// oaksLibrary/fbPumpMotion
// Block för global pumpmotion. V i blocket sätter internt i blocket den globala variabeln oaksGVL.bPumpMotion. 
// oaksGVL.bPumpMotion finns knuten i fbMotor och aktiverar pumpmotion om bPumpmotionConfig i respektive fbMotor-instans är till.
FUNCTION_BLOCK fbPumpMotion
VAR_INPUT
END_VAR
VAR_OUTPUT
	{attribute 'OPC.UA.DA' := '1'}
	V AT %M*  : BOOL; //Pumpmotion aktiv~wp:[trendoptions]i:14400, t:1
	{attribute 'OPC.UA.DA' := '1'}
	PV AT %M*  : STRING; //Dag för motionering~wp:
	{attribute 'OPC.UA.DA' := '1'}
	PV1 AT %M* : INT; //Tid för motionering~wp:[format]00:00
END_VAR
VAR
	stTime		: tc2_ba.TIMESTRUCT;
	nActualDayCase	: INT;
	nActualHour 	: INT;
	nActualMinute 	: INT;
	
	FB_BA_GetTime01 : tc2_ba.FB_BA_GetTime; 
	FB_BA_ExtTiSt01 : tc2_ba.FB_BA_ExtTiSt;	
	
	itemp : INT;
	nTime : INT; // Internvariabel aktuell tid (nActualHour+nActualMinute)
	
	bDay : BOOL; // Internvariabel blir TRUE om inställd dag är lika med aktuell dag
	bTime : BOOL; // Internvariabel blir TRUE om inställd tid är lika med aktuell tid
END_VAR
VAR_INPUT PERSISTENT
	{attribute 'OPC.UA.DA' := '1'}
	SP1 AT %M*  : INT:=1; //Dag för pumpmotion (0 = Söndag 1 = Måndag 2 = Tisdag..6 = Lördag~wp:
	{attribute 'OPC.UA.DA' := '1'}
	SP2 AT %M*  : INT:=1000; //Tid för pumpmotion~wp:[format]00:00[engmin]0[engmax]2400
END_VAR

	IF SP1 < 0 OR  SP1>6 THEN
		SP1 := 1;
	END_IF
	
	IF SP2 < 0 OR  SP2>2359 THEN
		SP2 := 1200;
	END_IF
	
	

	FB_BA_GetTime01(bEn :=TRUE);	
	stTime := FB_BA_GetTime01.stSysTi;

	nActualDayCase :=WORD_TO_INT (stTime.wDayOfWeek);
	nActualHour :=WORD_TO_INT (stTime.wHour)*100;
	nActualMinute :=WORD_TO_INT (stTime.wMinute);
	
	// nActualHour+nActualMinute
	
	nTime := nActualHour+nActualMinute;
	
	bDay := nActualDayCase = SP1;
	bTime := nTime = SP2;
	
	
	V := bDay AND bTime;
	
	oaksGVL.bPumpMotion := V;
	
	//För visning i Webport	
	PV1:= SP2;

	CASE SP1 OF
		0: PV:= 'Söndag';
		1: PV:= 'Måndag';
		2: PV:= 'Tisdag';
		3: PV:= 'Onsdag';
		4: PV:= 'Torsdag';
		5: PV:= 'Fredag';
		6: PV:= 'Lördag';
	END_CASE

END_FUNCTION_BLOCK

// oaksLibrary/Brand/fbFireDamperOneInput
//Funktionsblock för styrning av brandspjäll med stängt indikering (stänger på fjäder). 
FUNCTION_BLOCK fbFireDamperOneInput EXTENDS fbDigitalSignalLogic
VAR_INPUT
bMotion : BOOL; //Motionskörning
{attribute 'OPC.UA.DA' := '1'}
V2 AT %I* : BOOL; //Stängindikering~wp:[trendoptions]i:14400, t:1
END_VAR
VAR_OUTPUT
	{attribute 'OPC.UA.DA' := '1'}
	AL AT %M* : BOOL; //Spjällfel~wp:
	{attribute 'OPC.UA.DA' := '1'}
	PV4 AT %M* : BOOL; //Motionskörning aktiv~wp:[trendoptions]i:14400, t:1
END_VAR
VAR
	SR_1: SR;
	fbStartPulse: TP; // Startpuls	
	fbMotionTime: TP; // Håller en puls under motionskörning
	fbStopMotion: F_TRIG;
	TON_1: TON;
	bAlarm: BOOL;
END_VAR

SUPER^();
//Aktivera motionering på positiv flank (SET)
fbStartPulse(IN:= bMotion, PT:= T#1S, Q=> , ET=> ); //Startar en puls

//Hållkrets
SR_1(
SET1:= fbStartPulse.Q, 
RESET:= fbStopMotion.Q OR V2, 
Q1=> PV4
);

//Avaktivera motionering (RESET)
fbMotionTime(IN:= fbStartPulse.Q, PT:= T#180S, Q=> , ET=> ); //Startar en puls
fbStopMotion(CLK:= fbMotionTime.Q OR V2, Q=> ); // Reset då pulstid gått ut eller stängtindikering gått till

//Utgång
CMD := bSafe AND bStart AND NOT PV4;

//Larm
bAlarm := (NOT CMD AND NOT V2);
TON_1(IN:= bAlarm, PT:= T#30S, Q=> AL, ET=> );

END_FUNCTION_BLOCK

// oaksLibrary/Utsignal DO_AO/fbDigitalSignalLogic
// Block för digitala utsignaler med möjlighet att handställa utsignal. Larmar vid handställning.
FUNCTION_BLOCK fbDigitalSignalLogic
VAR_INPUT
	bStart : BOOL; // startvillkor
	bSafe: BOOL; // Säkerhetsvillkor
	bHandsetBlock : BOOL; // Används för blockering av handställning utan att blockera utsignal i autoläge. OBS! - För säkerhetsvillkor se ingång bSafe!
	tStartDelay : TIME := T#0S; // Startfördröjning
	tStopDelay : TIME := T#0S; // Stoppfördröjning
END_VAR
VAR_OUTPUT
	{attribute 'OPC.UA.DA' := '1'}
	CMD AT %Q* : BOOL; //Utsignal~wp:[trendoptions]i:14400, t:1
	{attribute 'OPC.UA.DA' := '1'}
	AL8 AT %M* : BOOL; //Utsignal handställd~wp:[alarmoptions]p:3
	STATE1 AT %M* : STRING; //Status IO-modul~wp:
	tStartDelayRemaining : TIME; // Aktuell  återstående tid startfördröjning
	tStopDelayRemaining : TIME; // Aktuell återstående tid toppfördröjning
END_VAR
VAR
	bInternalStart : BOOL;
	fbAlarm2 : fbAlarm; // Larm handställning
	//Handställningsvariabler från IO
	TI_bStateAuto AT %I* :BOOL :=TRUE; //Status Auto/Manuell
	TI_bStateRelay AT %I* :BOOL :=FALSE; //Status reläutgång
	bIOManual : BOOL;
	
	fbStartDelay: TON; // Startfördröjning
	fbStopDelay: TOF; // Stoppfördröjning
END_VAR
VAR_INPUT PERSISTENT
	{attribute 'OPC.UA.DA' := '1'}
	M AT %M* : BOOL; //Handställning~wp:[trendoptions]i:14400, t:1
	{attribute 'OPC.UA.DA' := '1'}
	MCMD AT %M* : BOOL; //Styrsignal handställning~wp:[trendoptions]i:14400, t:1
END_VAR

	//Handställning
	fbAlarm2(bInput:=M OR NOT TI_bStateAuto, tAlarmDelay:= , bAutoReset:=TRUE , bAlarmOutput=>AL8 );
	
	IF NOT bSafe OR bHandsetBlock THEN
		M := FALSE;
	END_IF;
	
	//Manuell omkopplare IO-modul
	bIOManual := fKx2652State(bAuto := TI_bStateAuto, bRelayStatus := TI_bStateRelay, sState => STATE1);
	
	
	//Start-/stoppfördröjning
    fbStartDelay(IN:=bStart , PT:=tStartDelay , Q=> , ET=> );
	fbStopDelay(IN:=fbStartDelay.Q, PT:=tStopDelay , Q=> , ET=> );
	
	tStopDelayRemaining := mTimeRemainingTof(fbStopDelay);
	tStartDelayRemaining := mTimeRemainingTon(fbStartDelay);
	
	bInternalStart := fbStopDelay.Q;
	
	IF NOT TI_bStateAuto THEN
		CMD := bIOManual;
	ELSE
		CMD := (((bInternalStart AND NOT M) OR (M AND MCMD)) AND bSafe) OR bIOManual;
	END_IF

METHOD PUBLIC mStartDelayRemaining : STRING
VAR_INPUT
	sStatusString : STRING;
END_VAR
VAR
	tTime : TIME; 
END_VAR
	tTime := mTimeRemainingTon(fbStartDelay);
	
	
	IF tTime > T#0S AND tTime < fbStartDelay.PT AND NOT M AND TI_bStateAuto  THEN
 		mStartDelayRemaining := CONCAT(sStatusString,CONCAT(INT_TO_STRING(TIME_TO_INT(tTime/1000)), ' s'));
	ELSE
		mStartDelayRemaining := ' ';
	END_IF
END_METHOD

METHOD PUBLIC mStopDelayRemaining : STRING
VAR_INPUT
	sStatusString : STRING;
END_VAR
VAR
	tTime : TIME; 
END_VAR
	tTime := mTimeRemainingTof(fbStopDelay);
	
	
	IF tTime > T#0S AND tTime < fbStopDelay.PT AND NOT M AND TI_bStateAuto  THEN
 		mStopDelayRemaining := CONCAT(sStatusString,CONCAT(INT_TO_STRING(TIME_TO_INT(tTime/1000)), ' s'));
	ELSE
		mStopDelayRemaining := ' ';
	END_IF
END_METHOD

METHOD PROTECTED mTimeRemainingTof : TIME
VAR_IN_OUT
	fbTof : TOF;
END_VAR
mTimeRemainingTof := fbTof.PT - fbTof.ET;
END_METHOD

METHOD PROTECTED mTimeRemainingTon : TIME
VAR_IN_OUT
	fbTon : TON;
END_VAR
mTimeRemainingTon := fbTon.PT - fbTon.ET;
END_METHOD

END_FUNCTION_BLOCK

// oaksLibrary/Brand/fbFireDamperWithAnalogOutput
//Oaks AB 2020-06-10
//Funktionsblock för styrning av brandspjäll med öppet/stängt indikering (stänger på fjäder). 
FUNCTION_BLOCK fbFireDamperWithAnalogOutput EXTENDS fbAnalogSignalLogic
VAR_INPUT
bMotion : BOOL; //Motionskörning
bSafe : BOOL; //Säkerhetsvillkor
tAlarmDelay : TIME := T#180S; // Larmfördröjning
END_VAR
VAR_OUTPUT
{attribute 'OPC.UA.DA' := '1'}
CMD AT %Q* : BOOL; //Manöver~wp:[trendoptions]i:14400, t:1
{attribute 'OPC.UA.DA' := '1'}
V0 AT %I* : BOOL; //Stängtindikering~wp:[trendoptions]i:14400, t:1
{attribute 'OPC.UA.DA' := '1'}
V1 AT %I* : BOOL; //Öppetindikering~wp:[trendoptions]i:14400, t:1
{attribute 'OPC.UA.DA' := '1'}
AL AT %M* : BOOL; //Spjällfel~wp:
{attribute 'OPC.UA.DA' := '1'}
PV4 AT %M* : BOOL; //Motionskörning aktiv~wp:[trendoptions]i:14400, t:1
END_VAR
VAR
	SR_1: SR;
	fbStartPulse: TP; // Startpuls	
	fbMotionTime: TP; // Håller en puls under motionskörning
	fbStopMotion: F_TRIG;
	fbAlarm1: fbAlarm;
	bAlarm: BOOL;
	IN: INT;
END_VAR

SUPER^();
//Aktivera motionering på positiv flank (SET)
fbStartPulse(IN:= bMotion, PT:= T#1S, Q=> , ET=> ); //Startar en puls
//Hållkrets
SR_1(
SET1:= fbStartPulse.Q, 
RESET:= fbStopMotion.Q OR V0, 
Q1=> PV4
);

//Avaktivera motionering (RESET)
fbMotionTime(IN:= fbStartPulse.Q, PT:= T#300S, Q=> , ET=> ); //Startar en puls
fbStopMotion(CLK:= fbMotionTime.Q, Q=> ); // Reset då pulstid gått ut

//Utgång
CMD := bSafe AND NOT PV4;

//Larm
bAlarm := (NOT CMD AND NOT V0) OR (CMD AND rSetpoint = 100 AND NOT V1);

fbAlarm1(bInput:=bAlarm , tAlarmDelay:=tAlarmDelay , bAutoReset:= TRUE, bAlarmOutput=> AL);

END_FUNCTION_BLOCK

// oaksLibrary/Utsignal DO_AO/fbAnalogSignalLogic
// Block för analoga utsignaler med möjlighet att handställa utsignal. Larmar vid handställning.
FUNCTION_BLOCK fbAnalogSignalLogic
VAR_INPUT
	rScaleX1 : REAL := 0; // Ändra om det är 2-10V exempelvis. Max är 0..32767 så 2-10V = 32767 * 0.2 = 6553
	rScaleX2 : REAL := 32767;
	rSetpoint : REAL; // Insginal för auto-läge (exmepelvis regulatorsignal)
	bInterlock : BOOL; // blockering av handställning
	bInvert : BOOL := FALSE; //Invertering utgång
END_VAR
VAR_OUTPUT
	{attribute 'OPC.UA.DA' := '1'}
	OP AT %M* : REAL;  //Utsignal~wp:[unit]%[format]0[trendoptions]i:300
	{attribute 'OPC.UA.DA' := '1'}
	AL8 AT %M* : BOOL;//Utsignal handställd~wp:[alarmoptions]p:3
END_VAR
VAR
	FB_BA_AO01 : FB_BA_AO;
	rY  AT %Q*: REAL;
	TO_iY AT %Q* : INT; 
	rOutputInternal : REAL; //Intern signal för invertering/ej invertering
	
	fbAlarm2 : fbAlarm; // Larm handställning
END_VAR
VAR_INPUT PERSISTENT
	{attribute 'OPC.UA.DA' := '1'}
	M AT %M*: BOOL;//Handställning~wp:[trendoptions]i:14400, t:1
	{attribute 'OPC.UA.DA' := '1'}
	OPM AT %M* : REAL;//Värde handställning~wp:[unit]%[format]0
END_VAR

	//Blockering handställning
	IF bInterlock THEN
		M := FALSE;
	END_IF;

	//Handställning
	IF M  THEN
		OP := OPM; 
	ELSE
		OP := rSetpoint;  
	END_IF
	
	//Handställningslarm
	fbAlarm2(bInput:=M , tAlarmDelay:= , bAutoReset:=TRUE , bAlarmOutput=>AL8 );
	
	//Invertering utång
	IF bInvert THEN
		rOutputInternal := (100 - OP);
	ELSE 
		rOutputInternal := OP;
	END_IF;		
		
	//Hantering utgång	
	FB_BA_AO01(
		rX:= rOutputInternal, 
		rX01:= 0, 
		rX02:= 100, 
		rY01:= rScaleX1, 
		rY02:= rScaleX2 , 
		udiOpMod:= , 
		rXManual:= , 
		rY=> rY, 
		TO_iY=>TO_iY );

END_FUNCTION_BLOCK

// oaksLibrary/Brand/fbSmokeDetector
// Block för rökdetektor med servicelarm.
FUNCTION_BLOCK fbSmokeDetector
VAR_INPUT
	{attribute 'OPC.UA.DA' := '1'}
	V3 AT %I* : BOOL; //Larmingång röklarm~wp:[trendoptions]i:14400, t:1
	bInvertedSmokeAlarm : BOOL; // invertering röklarm
	{attribute 'OPC.UA.DA' := '1'}
	V4 AT %I* : BOOL; //Larmingång servicelarm~wp:[trendoptions]i:14400, t:1
	bInvertedServiceAlarm : BOOL; // invertering servicelarm
	bAutoReset : BOOL := TRUE; // Auto-reset av larm
END_VAR
VAR_OUTPUT
	{attribute 'OPC.UA.DA' := '1'}
	AL AT %M* : BOOL; //Utlöst rökdetektor~wp:[alarmoptions]p:1
	{attribute 'OPC.UA.DA' := '1'}
	AL1 AT %M* : BOOL; //Servicelarm rökdetektor~wp:
END_VAR
VAR
	bInternalIndicationSmokeAlarm : BOOL;
	fbAlarmSmokeAlarm : fbAlarm;
	
	bInternalIndicationServiceAlarm : BOOL;
	fbAlarmServiceAlarm : fbAlarm;
END_VAR

	IF NOT bInvertedSmokeAlarm THEN
		bInternalIndicationSmokeAlarm :=  V3;
	ELSE
		bInternalIndicationSmokeAlarm := NOT V3;
	END_IF
		
	
	fbAlarmSmokeAlarm(
	bInput:= bInternalIndicationSmokeAlarm, 
	tAlarmDelay:= T#3S, 
	bAutoReset:= bAutoReset, 
	bAlarmOutput=>AL );
	
	IF NOT bInvertedServiceAlarm THEN
		bInternalIndicationServiceAlarm :=  V4;
	ELSE
		bInternalIndicationServiceAlarm := NOT V4;
	END_IF
		
	
	fbAlarmServiceAlarm(
	bInput:= bInternalIndicationServiceAlarm, 
	tAlarmDelay:= T#3S, 
	bAutoReset:= bAutoReset, 
	bAlarmOutput=>AL1 );

END_FUNCTION_BLOCK

// oaksLibrary/Börvärden/fbPowerLimiter
//Oaks AB
//2021-01-07
//Funktionsblock för effektbegräsning av temperatur för tex. VS/KB.
FUNCTION_BLOCK fbPowerLimiter
VAR_INPUT
	
	//Effektbegränsing
	rInstantaneousPower : REAL; //Momentaneffekt (kW)
	
END_VAR

VAR_OUTPUT
	
	//Effektbegränsning
	{attribute 'OPC.UA.DA' := '1'}
	PV AT %M* : REAL :=0; //Förskjutning från effektbegränsning~wp:[unit]°C[format]0.0
	{attribute 'OPC.UA.DA' := '1'}
	PV1 AT %M* : REAL :=0; //Momentaneffekt av max~wp:[unit]%[format]0
	{attribute 'OPC.UA.DA' := '1'}
	PV2 AT %M* : REAL :=0; //Max. energi per timme~wp:[unit]kWh[format]0
	{attribute 'OPC.UA.DA' := '1'}
	PV8 AT %M* : STRING; //Konfigurering~wp:
	{attribute 'OPC.UA.DA' := '1'}
	AL AT %M* : BOOL; //Effektbegränsning lång aktiveringstid~wp:[alarmoptions]p:2
	{attribute 'OPC.UA.DA' := '1'}
	V AT %M* : BOOL; //Effektbegränsning aktiv~wp:[trendoptions]i:14400, t:1
	
END_VAR

VAR

	rkWhMax : REAL;
	rLimitOffset : REAL; //Förskjutning från effektbegränsning
	rProcentOffMax : REAL; 
	
	fbAlarmLimit: fbAlarm;
	fbPowerLimiter : tc3_BA.FB_BA_Chrct02;
END_VAR

VAR_INPUT PERSISTENT
	
	//Effektstyrning
	{attribute 'OPC.UA.DA' := '1'}
	MO AT %M* : BOOL := FALSE; //Aktivering effektbegränsning~wp:[trendoptions]i:14400, t:1
	{attribute 'OPC.UA.DA' := '1'}
	SP1 AT %M* : REAL :=10000; //Max förbrukning per dygn~wp:[unit]kWh[format]0
	{attribute 'OPC.UA.DA' := '1'}
	SP2 AT %M* : REAL :=0; //Max förskjutning temperatur effekbegränsning~wp:[unit]°C[format]0.0
	{attribute 'OPC.UA.DA' := '1'}
	SP3 AT %M* : REAL :=90; //Min effektbegränsning då använd effekt >~wp:[unit]%[format]0
	{attribute 'OPC.UA.DA' := '1'}
	SP4 AT %M* : REAL :=95; //Max effektbegränsning då använd effekt >~wp:[unit]%[format]0
	{attribute 'OPC.UA.DA' := '1'}
	AD AT %M* : REAL :=24; //Larmfördröjning lång inkopplingstid effektbegränsning~wp:[unit]timmar[format]0
	
END_VAR

//Hantering ingångsvärden
IF SP1 < 0 THEN 
	SP1 := 0;
END_IF

IF SP3 > 100 OR SP3 < 0 THEN 
	SP1 := 95;
END_IF

IF SP4 < SP3 THEN
	SP4 := SP3 + 1;
END_IF

//Räkna ut momentanvärden
rkWhMax := SP1/24;
//Visning av energi per timme. 
PV2 := rkWhMax;

//Räkna ut procent av maxeffekt
IF rkWhMax > 0 THEN
	rProcentOffMax := rInstantaneousPower / rkWhMax;
	//Aktuell förbrukning i procent mot maxeffekt
	PV1 := rProcentOffMax * 100;
END_IF

//Konfigurering
IF SP2 = 0 THEN
	PV8 := 'Ej aktiv';
ELSIF SP2 < 0 THEN
	PV8 := 'Värmekrets (neg. förskj.)';
ELSIF SP2 > 0 THEN
	PV8 := 'Kylkrets (pos. förskj.)';
END_IF

//Aktiverad effektvakt
IF MO AND PV1 > SP3 AND SP2 <> 0 THEN
	V := TRUE;
ELSE 
	V := FALSE;
END_IF

fbPowerLimiter(
	rX:= rProcentOffMax, 
	rX01:= (SP3 * 0.01), 
	rX02:= (SP4 * 0.01), 
	rY01:= 0, 
	rY02:= SP2, 
	bLmt:= TRUE, 
	rY=> rLimitOffset, 
	bErr=> , 
	sErrDescr=> );

//Aktivering effektvakt
IF MO THEN
	PV := rLimitOffset;
ELSE
	PV := 0;
END_IF
	
//Lång inkopplingstid
fbAlarmLimit(bInput:= V, tAlarmDelay:= fRealToHour(AD), bAutoReset:= TRUE, bAlarmOutput=> AL);

END_FUNCTION_BLOCK

// oaksLibrary/Börvärden/fbRoomCompensation
//Rumskompensering med inställbar förskjutning per avvikande grad från börvärde
//Inställbar min / max begränsning på kompenseringen samt knapp för att aktivera
//V1.0 | JP 2024-07-16
FUNCTION_BLOCK fbRoomCompensation
VAR_INPUT
	PV AT %M*: REAL; //Aktuell temperatur~wp:[unit]°C[format]0.0[trendoption]i:300
END_VAR
VAR_OUTPUT
	CSP AT %M*: REAL; //Börvärdesförskjutning~wp:[unit]°C[format]0.0[trendoption]i:300
	V AT %M* : BOOL; //Indikering aktiv rumskompensering~wp:
END_VAR
VAR
	rTempAvgDiff: REAL;
	rTempZeroPoint: REAL;
	rMellanInnanUt: REAL;
END_VAR
VAR PERSISTENT
	MO AT %M* : BOOL; //Aktivering av rumskompensering~wp:
	SP AT %M*: REAL := 21; //Rumsbörvärde~wp:[unit]°C[format]0.0
	SP1 AT %M*: REAL := 3; //Pararellförskjutning per minusgrad~wp:[unit]°C[format]0.0
	SP2 AT %M*: REAL := -3; //Pararellförskjutning per plusgrad~wp:[unit]°C[format]0.0
	SP3 AT %M*: REAL := -6; //Lägsta tillåtna förskjutning~wp:[unit]°C[format]0.0
	SP4 AT %M*: REAL := 6; //Högsta tillåtna förskjutning~wp:[unit]°C[format]0.0
END_VAR

rTempAvgDiff := SP - PV;	
	
	rTempZeroPoint := rTempAvgDiff;
	
	IF (rTempZeroPoint>=0) THEN
		//Increase
		rMellanInnanUt := (rTempZeroPoint * SP1);
	ELSE 
		//Decrease
		rMellanInnanUt := (0 -(rTempZeroPoint * SP2));
	END_IF
	
IF MO THEN
	CSP:=LIMIT(SP3, rMellanInnanUt, SP4);
ELSE
	CSP:= 0;
END_IF

IF MO AND CSP <> 0 THEN
	V:= TRUE;
ELSE 
	V:= FALSE;
END_IF

END_FUNCTION_BLOCK

// oaksLibrary/Börvärden/fbSetPointBase
//Oaks AB
//2020-09-07
//Funktionsblock för hantering av börvärde från internt och från överordnat system. Basblock
FUNCTION_BLOCK fbSetPointBase 

VAR_INPUT
	rISP : REAL; //Internt börvärde/offset då M=1
	bISPconfig : BOOL :=FALSE; //False=Absolutbörvärde True=Offset då M=1
	bISPcomError : BOOL :=FALSE; //Kommunikationsfel då M=1
	rPowerLimitOffset : REAL := 0; //Förskjutning från effektbegränsning
	rSetpointOffset : REAL := 0; // Börvärdesförskjutning då M = 0.
END_VAR

VAR_OUTPUT
	{attribute 'OPC.UA.DA' := '1'}
	FAULT AT %M* : BOOL; //Kommunikationsfel från överordnat system~wp:[alarmoptions]p:2
	
END_VAR

VAR
	//Börvärde
	rISPinternal : REAL;
	rSetPoint : REAL ; //Internt börvärde
	rCsp : REAL; //Uträknat börvärde
	rESP : REAL; //Externt börvärde
	rMin : REAL; //Intern minbegränsning
	rMax : REAL; //Intern maxbegränsning
	
	fbToggle_1: fbToggle;
	fbAlarm: fbAlarm;
	{attribute 'OPC.UA.DA' := '1'}
	V3 AT %M* : BOOL :=FALSE; //Watchdog sätts till 1 varje 15 minut~wp:
	{attribute 'OPC.UA.DA' := '1'}
	PV1 AT %M* : STRING :=''; //Källa börvärde~wp:
	
	powerLimiterStatus : STRING; 
	bSetpointTypeBase : STRING :='';
		
END_VAR

VAR_INPUT PERSISTENT
	{attribute 'OPC.UA.DA' := '1'}
	M AT %M* : INT :=0; //Källa börvärde 0=Internt börvärde/kurva/1=Optimering/2=Externt börvärde~wp:	
END_VAR

//Vakthund endast vid driftfall Extern
	//Sätt indikering till noll var varje minut
	fbToggle_1(bStart:= (M = 2), tTimeOn:= T#1M, tTimeOff:= T#1s, bOutput=> );
	IF fbToggle_1.bOutput = TRUE THEN
		V3 := FALSE;
	END_IF
	
	//Skapa larm om inte värde satts till 1
	IF M = 2 AND NOT V3 THEN
		fbalarm.bInput := TRUE;
	ELSE
		fbalarm.bInput := FALSE;
	END_IF
		
		fbAlarm(bInput:= , tAlarmDelay:= T#30M, bAutoReset:= TRUE, bAlarmOutput=> FAULT);
	
	//Börvärdestyp på intern börvärdesförskjutning
	IF bISPconfig THEN	
		rISPinternal := rISP + rSetPoint;
	ELSE
		rISPinternal := rISP;
	END_IF
		
//Effektbegränsning
IF rPowerLimitOffset <> 0 THEN
	powerLimiterStatus := ' / Aktiv effektbegränsning';
ELSE
	powerLimiterStatus := '';
END_IF		
		
//Hantering av larm och driftläge	
	IF M = 1 THEN
		IF bISPcomError THEN
			//Vid komm.fel använd internt börvärde och sätt felindikering	
			rCsp := rCsp := LIMIT(rMin,(rSetPoint + rPowerLimitOffset + rSetpointOffset),rMax);
			PV1 := 'Komm.fel, internt börvärde används';
		ELSE
			//Annars använd ingångsvärde
			rCsp := LIMIT(rMin,(rISPinternal + rPowerLimitOffset),rMax);
			PV1 := CONCAT('Optimering',powerLimiterStatus);
		END_IF;
		
	ELSIF M = 2 AND NOT FAULT THEN
		rCsp := LIMIT(rMin,(rESP + rPowerLimitOffset),rMax);
		PV1 := CONCAT('Externt börvärde',powerLimiterStatus);
	
	ELSE
		rCsp := LIMIT(rMin,(rSetPoint + rPowerLimitOffset + rSetpointOffset),rMax);
		PV1 := CONCAT(bSetpointTypeBase,powerLimiterStatus);
	END_IF;

END_FUNCTION_BLOCK

// oaksLibrary/Börvärden/fbSetPointC
//Oaks AB
//2020-09-07
//Funktionsblock med inbyggt börvärde och börvärdeförskjutning.
FUNCTION_BLOCK fbSetPointC EXTENDS fbSetPointBase

VAR_INPUT PERSISTENT
	{attribute 'OPC.UA.DA' := '1'}
	SP AT %M* :  REAL:=56;	//Börvärde~wp:[unit]°C[format]0.0
	{attribute 'OPC.UA.DA' := '1'}
	ESP AT %M* : REAL:=0; //Externt börvärde (Absolutbörvärde)~wp:[unit]°C[format]0.0
END_VAR

VAR_OUTPUT
	{attribute 'OPC.UA.DA' := '1'}
	CSP AT %M*: REAL; //Uträknat börvärde~wp:[unit]°C[format]0.0
	{attribute 'OPC.UA.DA' := '1'}
	ISP AT %M* : REAL:=0; //Börvärde från optimering~wp:[unit]°C[format]0.0
		
END_VAR

	SUPER^(); 
	//Börvärde 
	rSetpoint := SP;
	
	//Läs från bas	
	CSP := rCSP;
	ISP := rIspInternal;
	//Skriv till bas
	rMin := MIN(ISP, SP, ESP) + rPowerLimitOffset;
	rMax := MAX(ISP,SP, ESP) + rPowerLimitOffset;
	rESP := ESP;
	bSetpointTypeBase := 'Internt börvärde';

END_FUNCTION_BLOCK

// oaksLibrary/Börvärden/fbSetPointCMinMax
//Oaks AB
//2020-09-07
//Funktionsblock med inbyggt börvärde och börvärdeförskjutning.
FUNCTION_BLOCK fbSetPointCMinMax EXTENDS fbSetPointBase

VAR_INPUT PERSISTENT
	{attribute 'OPC.UA.DA' := '1'}
	SP AT %M* :  REAL:=56;	//Börvärde~wp:[unit]°C[format]0.0
	{attribute 'OPC.UA.DA' := '1'}
	ESP AT %M* : REAL:=0; //Externt börvärde (Absolutbörvärde)~wp:[unit]°C[format]0.0
	{attribute 'OPC.UA.DA' := '1'}
	MN AT %M* :	REAL:=20; //Min.begränsning börvärde~wp:[unit]°C[format]0
	{attribute 'OPC.UA.DA' := '1'}
	MX AT %M* :	REAL:=65; //Max.begränsning börvärde~wp:[unit]°C[format]0
END_VAR

VAR_OUTPUT
	{attribute 'OPC.UA.DA' := '1'}
	CSP AT %M*: REAL; //Uträknat börvärde~wp:[unit]°C[format]0.0
	{attribute 'OPC.UA.DA' := '1'}
	ISP AT %M* : REAL:=0; //Börvärde från optimering~wp:[unit]°C[format]0.0
		
END_VAR

	SUPER^(); 
	//Börvärde 
	rSetpoint := SP;
	
	//Läs från bas	
	CSP := rCSP;
	ISP := rIspInternal;
	//Skriv till bas
	
	//Hantering min-max
	IF MN > SP THEN
		MN := SP - 1;
	END_IF
	
	IF MX < SP THEN
		MX := SP + 1;
	END_IF
		
	rMin := MN;
	rMax := MX;
	rESP := ESP;
	bSetpointTypeBase := 'Internt börvärde';

END_FUNCTION_BLOCK

// oaksLibrary/Börvärden/fbSetPointKpa
//Oaks AB
//2020-09-07
//Funktionsblock med inbyggt börvärde och börvärdeförskjutning.
FUNCTION_BLOCK fbSetPointKpa EXTENDS fbSetPointBase

VAR_INPUT PERSISTENT
	{attribute 'OPC.UA.DA' := '1'}
	SP AT %M* :  REAL:=56;	//Börvärde~wp:[unit]kPa[format]0
	{attribute 'OPC.UA.DA' := '1'}
	ESP AT %M* : REAL:=0; //Externt börvärde (Absolutbörvärde)~wp:[unit]kPa[format]0
END_VAR

VAR_OUTPUT
	{attribute 'OPC.UA.DA' := '1'}
	CSP AT %M*: REAL; //Uträknat börvärde~wp:[unit]kPa[format]0
	{attribute 'OPC.UA.DA' := '1'}
	ISP AT %M* : REAL:=0; //Börvärde från optimering~wp:[unit]kPa[format]0
		
END_VAR

	SUPER^(); 
	//Börvärde 
	rSetpoint := SP;
	
	//Läs från bas	
	CSP := rCSP;
	ISP := rIspInternal;
	//Skriv till bas
	rMin := MIN(ISP, SP, ESP) + rPowerLimitOffset;
	rMax := MAX(ISP,SP, ESP) + rPowerLimitOffset;
	rESP := ESP;
	bSetpointTypeBase := 'Internt börvärde';

END_FUNCTION_BLOCK

// oaksLibrary/Börvärden/fbSetPointLs
//Oaks AB
//2020-09-07
//Funktionsblock med inbyggt börvärde och börvärdeförskjutning.
FUNCTION_BLOCK fbSetPointLs EXTENDS fbSetPointBase

VAR_INPUT PERSISTENT
	{attribute 'OPC.UA.DA' := '1'}
	SP AT %M* :  REAL:=200;	//Börvärde~wp:[unit]l/s[format]0
	{attribute 'OPC.UA.DA' := '1'}
	ESP AT %M* : REAL:=0; //Externt börvärde (Absolutbörvärde)~wp:[unit]l/s[format]0
END_VAR

VAR_OUTPUT
	{attribute 'OPC.UA.DA' := '1'}
	CSP AT %M*: REAL; //Uträknat börvärde~wp:[unit]l/s[format]0
	{attribute 'OPC.UA.DA' := '1'}
	ISP AT %M* : REAL:=0; //Börvärde från optimering~wp:[unit]l/s[format]0
END_VAR

	SUPER^(); 
	//Börvärde
	rSetpoint := SP;
	
	//Läs från bas	
	CSP := rCSP;
	ISP := rIspInternal;
	//Skriv till bas
	rMin := MIN(ISP, SP, ESP) + rPowerLimitOffset;
	rMax := MAX(ISP,SP, ESP) + rPowerLimitOffset;
	rESP := ESP;
	bSetpointTypeBase := 'Internt börvärde';

END_FUNCTION_BLOCK

// oaksLibrary/Börvärden/fbSetPointOutdoorCompC
//Oaks AB
//2020-09-07
//Funktionsblock med inbyggd utekompensering och börvärdeförskjutning.
FUNCTION_BLOCK fbSetPointOutdoorCompC EXTENDS fbSetPointBase

VAR_INPUT
	rOutdoorTemperature : ANY; //Utetemperatur Knyter man inget här används oaksGVL.rOutdoortemp
	bOverrideCsp : BOOL := FALSE; //Aktivera direkt skrivning till CSP (Ex. nattkyla)
	rOverrideSetpoint: REAL := 0; // 
END_VAR	
VAR
	rTempUsed : REAL; // Uteluftstemperatur
	bAktiveraSkrivningCsp : BOOL := TRUE; // Aktiverar skrivning från detta block. Sätts till false om man vill använda detta blocket extendat och skriva från det extendade blocket.
END_VAR
VAR_INPUT PERSISTENT
	{attribute 'OPC.UA.DA' := '1'}
	Y1 AT %M* :  REAL:=60; //Utetemp/Börvärde~wp:[unit]°C[format]0.0
	{attribute 'OPC.UA.DA' := '1'}
	Y2 AT %M* :	REAL:=55; //Utetemp/Börvärde~wp:[unit]°C[format]0.0
	{attribute 'OPC.UA.DA' := '1'}
	Y3 AT %M* :	REAL:=50; //Utetemp/Börvärde~wp:[unit]°C[format]0.0
	{attribute 'OPC.UA.DA' := '1'}
	Y4 AT %M* :	REAL:=40; //Utetemp/Börvärde~wp:[unit]°C[format]0.0
	{attribute 'OPC.UA.DA' := '1'}
	Y5 AT %M* :	REAL:=30; //Utetemp/Börvärde~wp:[unit]°C[format]0.0
	{attribute 'OPC.UA.DA' := '1'}
	Y6 AT %M* :	REAL:=20; //Utetemp/Börvärde~wp:[unit]°C[format]0.0
	{attribute 'OPC.UA.DA' := '1'}
	X1 AT %M* :	REAL:=-30; //Utetemperatur~wp:[unit]°C[format]0.0
	{attribute 'OPC.UA.DA' := '1'}
	X2 AT %M* :	REAL:=-20; //Utetemperatur~wp:[unit]°C[format]0.0
	{attribute 'OPC.UA.DA' := '1'}
	X3 AT %M* :	REAL:=-10; //Utetemperatur~wp:[unit]°C[format]0.0
	{attribute 'OPC.UA.DA' := '1'}
	X4 AT %M* :	REAL:=0; //Utetemperatur~wp:[unit]°C[format]0.0
	{attribute 'OPC.UA.DA' := '1'}
	X5 AT %M* :	REAL:=10; //Utetemperatur~wp:[unit]°C[format]0.0
	{attribute 'OPC.UA.DA' := '1'}
	X6 AT %M* :	REAL:=20; //Utetemperatur~wp:[unit]°C[format]0.0
	{attribute 'OPC.UA.DA' := '1'}
	MN AT %M* :	REAL:=20; //Min.begränsning börvärde~wp:[unit]°C[format]0.0
	{attribute 'OPC.UA.DA' := '1'}
	MX AT %M* :	REAL:=65; //Max.begränsning börvärde~wp:[unit]°C[format]0.0
	{attribute 'OPC.UA.DA' := '1'}
	ESP AT %M* : REAL:=0; //Externt börvärde (Absolutbörvärde)~wp:[unit]°C[format]0.0
END_VAR

VAR_OUTPUT
	{attribute 'OPC.UA.DA' := '1'}
	CSP AT %M*: REAL; //Uträknat börvärde~wp:[unit]°C[format]0.0
	{attribute 'OPC.UA.DA' := '1'}
	ISP AT %M* : REAL:=0; //Börvärde från optimering~wp:[unit]°C[format]0.0
END_VAR

	SUPER^(); 
	//Temp select
	rTempUsed := F_GetTempToUse(rOutdoorTemperature);

	
	//Uträknat börvärde
	rSetpoint := fScale6p(
	rX:= rTempUsed, 
	Y1:= Y1, 
	Y2:= Y2, 
	Y3:= Y3, 
	Y4:= Y4, 
	Y5:= Y5, 
	Y6:= Y6, 
	X1:= X1, 
	X2:= X2, 
	X3:= X3, 
	X4:= X4, 
	X5:= X5, 
	X6:= X6);
	

	//Avvaktivera skrivning om M=0 och tex. nattkyla är aktiverad
	IF M = 0 AND bOverrideCsp THEN
		bAktiveraSkrivningCsp := FALSE; // Inaktivera skrivning i basblock för att kunna skriva csp från detta block.
		CSP := rOverrideSetpoint;
		bSetpointTypeBase := 'Intern kurva överstyrd';
	ELSE 
		bAktiveraSkrivningCsp := TRUE; // Inaktivera skrivning i basblock för att kunna skriva csp från detta block.
		bSetpointTypeBase := 'Intern kurva';
	END_IF
 	
	mBv(bAktiveraSkrivningCsp);

METHOD PROTECTED mBv : BOOL
VAR_INPUT
	bWriteCsp : BOOL;
END_VAR
		//Läs från bas	
		IF bWriteCsp THEN
			CSP := rCSP;
		END_IF;
		ISP := rIspInternal;
		//Skriv till bas
		rMin := MN;
		rMax := MX;
		rESP := ESP;
END_METHOD

END_FUNCTION_BLOCK

// oaksLibrary/Börvärden/fbSetPointOutdoorCompkPa
//Oaks AB
//2020-09-07
//Funktionsblock med inbyggd utekompensering och börvärdeförskjutning.
FUNCTION_BLOCK fbSetPointOutdoorCompkPa EXTENDS fbSetPointBase
VAR_INPUT
	rOutdoorTemperature : ANY; //Utetemperatur Knyter man inget här används oaksGVL.rOutdoortemp
	bOverrideCsp : BOOL := FALSE; //Aktivera direkt skrivning till CSP (Ex. nattkyla)
	rOverrideSetpoint: REAL := 0; // 
END_VAR	
VAR
	bAktiveraSkrivningCsp : BOOL := TRUE; // Aktiverar skrivning från detta block. Sätts till false om man vill använda detta blocket extendat och skriva från det extendade blocket.
	rTempUsed : REAL; // Uteluftstemperatur
END_VAR

VAR_INPUT PERSISTENT
	{attribute 'OPC.UA.DA' := '1'}
	Y1 AT %M* :  REAL:=60; //Utetemp/Börvärde~wp:[unit]kPa[format]0
	{attribute 'OPC.UA.DA' := '1'}
	Y2 AT %M* :	REAL:=55; //Utetemp/Börvärde~wp:[unit]kPa[format]0
	{attribute 'OPC.UA.DA' := '1'}
	Y3 AT %M* :	REAL:=50; //Utetemp/Börvärde~wp:[unit]kPa[format]0
	{attribute 'OPC.UA.DA' := '1'}
	Y4 AT %M* :	REAL:=40; //Utetemp/Börvärde~wp:[unit]kPa[format]0
	{attribute 'OPC.UA.DA' := '1'}
	Y5 AT %M* :	REAL:=30; //Utetemp/Börvärde~wp:[unit]kPa[format]0
	{attribute 'OPC.UA.DA' := '1'}
	Y6 AT %M* :	REAL:=20; //Utetemp/Börvärde~wp:[unit]kPa[format]0
	{attribute 'OPC.UA.DA' := '1'}
	X1 AT %M* :	REAL:=-30; //Utetemperatur~wp:[unit]°C[format]0.0
	{attribute 'OPC.UA.DA' := '1'}
	X2 AT %M* :	REAL:=-20; //Utetemperatur~wp:[unit]°C[format]0.0
	{attribute 'OPC.UA.DA' := '1'}
	X3 AT %M* :	REAL:=-10; //Utetemperatur~wp:[unit]°C[format]0.0
	{attribute 'OPC.UA.DA' := '1'}
	X4 AT %M* :	REAL:=0; //Utetemperatur~wp:[unit]°C[format]0.0
	{attribute 'OPC.UA.DA' := '1'}
	X5 AT %M* :	REAL:=10; //Utetemperatur~wp:[unit]°C[format]0.0
	{attribute 'OPC.UA.DA' := '1'}
	X6 AT %M* :	REAL:=20; //Utetemperatur~wp:[unit]°C[format]0.0
	{attribute 'OPC.UA.DA' := '1'}
	MN AT %M* :	REAL:=50; //Min.begränsning börvärde~wp:[unit]kPa[format]0
	{attribute 'OPC.UA.DA' := '1'}
	MX AT %M* :	REAL:=100; //Max.begränsning börvärde~wp:[unit]kPa[format]0
	{attribute 'OPC.UA.DA' := '1'}
	ESP AT %M* : REAL:=0; //Externt börvärde (Absolutbörvärde)~wp:[unit]kPa[format]0
END_VAR

VAR_OUTPUT
	{attribute 'OPC.UA.DA' := '1'}
	CSP AT %M*: REAL; //Uträknat börvärde~wp:[unit]kPa[format]0
	{attribute 'OPC.UA.DA' := '1'}
	ISP AT %M* : REAL:=0; //Börvärde från optimering~wp:[unit]kPa[format]0
END_VAR

	SUPER^(); 
	//Temp select
	rTempUsed := F_GetTempToUse(rOutdoorTemperature);

	
	//Uträknat börvärde
	rSetpoint := fScale6p(
	rX:= rTempUsed, 
	Y1:= Y1, 
	Y2:= Y2, 
	Y3:= Y3, 
	Y4:= Y4, 
	Y5:= Y5, 
	Y6:= Y6, 
	X1:= X1, 
	X2:= X2, 
	X3:= X3, 
	X4:= X4, 
	X5:= X5, 
	X6:= X6);
	

	//Avvaktivera skrivning om M=0 och tex. nattkyla är aktiverad
	IF M = 0 AND bOverrideCsp THEN
		bAktiveraSkrivningCsp := FALSE; // Inaktivera skrivning i basblock för att kunna skriva csp från detta block.
		CSP := rOverrideSetpoint;
		bSetpointTypeBase := 'Intern kurva överstyrd';
	ELSE 
		bAktiveraSkrivningCsp := TRUE; // Inaktivera skrivning i basblock för att kunna skriva csp från detta block.
		bSetpointTypeBase := 'Intern kurva';
	END_IF
	
	mBv(bAktiveraSkrivningCsp);

METHOD PROTECTED mBv : BOOL
VAR_INPUT
	bWriteCsp : BOOL;
END_VAR
		//Läs från bas	
		IF bWriteCsp THEN
			CSP := rCSP;
		END_IF;
		ISP := rIspInternal;
		//Skriv till bas
		rMin := MN;
		rMax := MX;
		rESP := ESP;
END_METHOD

END_FUNCTION_BLOCK

// oaksLibrary/Börvärden/fbSetPointOutdoorCompLs
//Oaks AB
//2020-09-07
//Funktionsblock med inbyggd utekompensering och börvärdeförskjutning.
FUNCTION_BLOCK fbSetPointOutdoorCompLs EXTENDS fbSetPointBase
VAR_INPUT
	rOutdoorTemperature : ANY; //Utetemperatur Knyter man inget här används oaksGVL.rOutdoortemp
	bOverrideCsp : BOOL := FALSE; //Aktivera direkt skrivning till CSP (Ex. nattkyla)
	rOverrideSetpoint: REAL := 0; // 
END_VAR	
VAR
	bAktiveraSkrivningCsp : BOOL := TRUE; // Aktiverar skrivning från detta block. Sätts till false om man vill använda detta blocket extendat och skriva från det extendade blocket.
	rTempUsed : REAL; // Uteluftstemperatur
END_VAR

VAR_INPUT PERSISTENT
	{attribute 'OPC.UA.DA' := '1'}
	Y1 AT %M* :  REAL:=60; //Utetemp/Börvärde~wp:[unit]l/s[format]0
	{attribute 'OPC.UA.DA' := '1'}
	Y2 AT %M* :	REAL:=55; //Utetemp/Börvärde~wp:[unit]l/s[format]0
	{attribute 'OPC.UA.DA' := '1'}
	Y3 AT %M* :	REAL:=50; //Utetemp/Börvärde~wp:[unit]l/s[format]0
	{attribute 'OPC.UA.DA' := '1'}
	Y4 AT %M* :	REAL:=40; //Utetemp/Börvärde~wp:[unit]l/s[format]0
	{attribute 'OPC.UA.DA' := '1'}
	Y5 AT %M* :	REAL:=30; //Utetemp/Börvärde~wp:[unit]l/s[format]0
	{attribute 'OPC.UA.DA' := '1'}
	Y6 AT %M* :	REAL:=20; //Utetemp/Börvärde~wp:[unit]l/s[format]0
	{attribute 'OPC.UA.DA' := '1'}
	X1 AT %M* :	REAL:=-30; //Utetemperatur~wp:[unit]°C[format]0.0
	{attribute 'OPC.UA.DA' := '1'}
	X2 AT %M* :	REAL:=-20; //Utetemperatur~wp:[unit]°C[format]0.0
	{attribute 'OPC.UA.DA' := '1'}
	X3 AT %M* :	REAL:=-10; //Utetemperatur~wp:[unit]°C[format]0.0
	{attribute 'OPC.UA.DA' := '1'}
	X4 AT %M* :	REAL:=0; //Utetemperatur~wp:[unit]°C[format]0.0
	{attribute 'OPC.UA.DA' := '1'}
	X5 AT %M* :	REAL:=10; //Utetemperatur~wp:[unit]°C[format]0.0
	{attribute 'OPC.UA.DA' := '1'}
	X6 AT %M* :	REAL:=20; //Utetemperatur~wp:[unit]°C[format]0.0
	{attribute 'OPC.UA.DA' := '1'}
	MN AT %M* :	REAL:=20; //Min.begränsning börvärde~wp:[unit]l/s[format]0
	{attribute 'OPC.UA.DA' := '1'}
	MX AT %M* :	REAL:=65; //Max.begränsning börvärde~wp:[unit]l/s[format]0
	{attribute 'OPC.UA.DA' := '1'}
	ESP AT %M* : REAL:=0; //Externt börvärde (Absolutbörvärde)~wp:[unit]l/s[format]0
END_VAR

VAR_OUTPUT
	{attribute 'OPC.UA.DA' := '1'}
	CSP AT %M*: REAL; //Uträknat börvärde~wp:[unit]l/s[format]0
	{attribute 'OPC.UA.DA' := '1'}
	ISP AT %M* : REAL:=0; //Börvärde från optimering~wp:[unit]l/s[format]0
END_VAR

	SUPER^(); 
	//Temp select
	rTempUsed := F_GetTempToUse(rOutdoorTemperature);
	//Uträknat börvärde
	rSetpoint := fScale6p(
	rX:= rTempUsed, 
	Y1:= Y1, 
	Y2:= Y2, 
	Y3:= Y3, 
	Y4:= Y4, 
	Y5:= Y5, 
	Y6:= Y6, 
	X1:= X1, 
	X2:= X2, 
	X3:= X3, 
	X4:= X4, 
	X5:= X5, 
	X6:= X6);
	
	//Avvaktivera skrivning om M=0 och tex. nattkyla är aktiverad
	IF M = 0 AND bOverrideCsp THEN
		bAktiveraSkrivningCsp := FALSE; // Inaktivera skrivning i basblock för att kunna skriva csp från detta block.
		CSP := rOverrideSetpoint;
		bSetpointTypeBase := 'Intern kurva överstyrd';
	ELSE 
		bAktiveraSkrivningCsp := TRUE; // Inaktivera skrivning i basblock för att kunna skriva csp från detta block.
		bSetpointTypeBase := 'Intern kurva';
	END_IF
	
	mBv(bAktiveraSkrivningCsp);

METHOD PROTECTED mBv : BOOL
VAR_INPUT
	bWriteCsp : BOOL;
END_VAR
		//Läs från bas	
		IF bWriteCsp THEN
			CSP := rCSP;
		END_IF;
		ISP := rIspInternal;
		//Skriv till bas
		rMin := MN;
		rMax := MX;
		rESP := ESP;
END_METHOD

END_FUNCTION_BLOCK

// oaksLibrary/Börvärden/fbSetPointOutdoorCompPa
//Oaks AB
//2020-09-07
//Funktionsblock med inbyggd utekompensering och börvärdeförskjutning.
FUNCTION_BLOCK fbSetPointOutdoorCompPa EXTENDS fbSetPointBase
VAR_INPUT
	rOutdoorTemperature : ANY; //Utetemperatur Knyter man inget här används oaksGVL.rOutdoortemp
	bOverrideCsp : BOOL := FALSE; //Aktivera direkt skrivning till CSP (Ex. nattkyla)
	rOverrideSetpoint: REAL := 0; // 
END_VAR	
VAR
	bAktiveraSkrivningCsp : BOOL := TRUE; // Aktiverar skrivning från detta block. Sätts till false om man vill använda detta blocket extendat och skriva från det extendade blocket.
	rTempUsed : REAL; // Uteluftstemperatur
END_VAR

VAR_INPUT PERSISTENT
	{attribute 'OPC.UA.DA' := '1'}
	Y1 AT %M* :  REAL:=60; //Utetemp/Börvärde~wp:[unit]Pa[format]0
	{attribute 'OPC.UA.DA' := '1'}
	Y2 AT %M* :	REAL:=55; //Utetemp/Börvärde~wp:[unit]Pa[format]0
	{attribute 'OPC.UA.DA' := '1'}
	Y3 AT %M* :	REAL:=50; //Utetemp/Börvärde~wp:[unit]Pa[format]0
	{attribute 'OPC.UA.DA' := '1'}
	Y4 AT %M* :	REAL:=40; //Utetemp/Börvärde~wp:[unit]Pa[format]0
	{attribute 'OPC.UA.DA' := '1'}
	Y5 AT %M* :	REAL:=30; //Utetemp/Börvärde~wp:[unit]Pa[format]0
	{attribute 'OPC.UA.DA' := '1'}
	Y6 AT %M* :	REAL:=20; //Utetemp/Börvärde~wp:[unit]Pa[format]0
	{attribute 'OPC.UA.DA' := '1'}
	X1 AT %M* :	REAL:=-30; //Utetemperatur~wp:[unit]°C[format]0.0
	{attribute 'OPC.UA.DA' := '1'}
	X2 AT %M* :	REAL:=-20; //Utetemperatur~wp:[unit]°C[format]0.0
	{attribute 'OPC.UA.DA' := '1'}
	X3 AT %M* :	REAL:=-10; //Utetemperatur~wp:[unit]°C[format]0.0
	{attribute 'OPC.UA.DA' := '1'}
	X4 AT %M* :	REAL:=0; //Utetemperatur~wp:[unit]°C[format]0.0
	{attribute 'OPC.UA.DA' := '1'}
	X5 AT %M* :	REAL:=10; //Utetemperatur~wp:[unit]°C[format]0.0
	{attribute 'OPC.UA.DA' := '1'}
	X6 AT %M* :	REAL:=20; //Utetemperatur~wp:[unit]°C[format]0.0
	{attribute 'OPC.UA.DA' := '1'}
	MN AT %M* :	REAL:=50; //Min.begränsning börvärde~wp:[unit]Pa[format]0
	{attribute 'OPC.UA.DA' := '1'}
	MX AT %M* :	REAL:=100; //Max.begränsning börvärde~wp:[unit]Pa[format]0
	{attribute 'OPC.UA.DA' := '1'}
	ESP AT %M* : REAL:=0; //Externt börvärde (Absolutbörvärde)~wp:[unit]Pa[format]0
END_VAR

VAR_OUTPUT
	{attribute 'OPC.UA.DA' := '1'}
	CSP AT %M*: REAL; //Uträknat börvärde~wp:[unit]Pa[format]0
	{attribute 'OPC.UA.DA' := '1'}
	ISP AT %M* : REAL:=0; //Börvärde från optimering~wp:[unit]Pa[format]0
END_VAR

	SUPER^(); 
	//Temp select
	rTempUsed := F_GetTempToUse(rOutdoorTemperature);

	
	//Uträknat börvärde
	rSetpoint := fScale6p(
	rX:= rTempUsed, 
	Y1:= Y1, 
	Y2:= Y2, 
	Y3:= Y3, 
	Y4:= Y4, 
	Y5:= Y5, 
	Y6:= Y6, 
	X1:= X1, 
	X2:= X2, 
	X3:= X3, 
	X4:= X4, 
	X5:= X5, 
	X6:= X6);
	
	//Avvaktivera skrivning om M=0 och tex. nattkyla är aktiverad
	IF M = 0 AND bOverrideCsp THEN
		bAktiveraSkrivningCsp := FALSE; // Inaktivera skrivning i basblock för att kunna skriva csp från detta block.
		CSP := rOverrideSetpoint;
		bSetpointTypeBase := 'Intern kurva överstyrd';
	ELSE 
		bAktiveraSkrivningCsp := TRUE; // Inaktivera skrivning i basblock för att kunna skriva csp från detta block.
		bSetpointTypeBase := 'Intern kurva';
	END_IF
	
	mBv(bAktiveraSkrivningCsp);

METHOD PROTECTED mBv : BOOL
VAR_INPUT
	bWriteCsp : BOOL;
END_VAR
		//Läs från bas	
		IF bWriteCsp THEN
			CSP := rCSP;
		END_IF;
		ISP := rIspInternal;
		//Skriv till bas
		rMin := MN;
		rMax := MX;
		rESP := ESP;
END_METHOD

END_FUNCTION_BLOCK

// oaksLibrary/Börvärden/fbSetPointPa
//Oaks AB
//2020-09-07
//Funktionsblock med inbyggt börvärde och börvärdeförskjutning.
FUNCTION_BLOCK fbSetPointPa EXTENDS fbSetPointBase

VAR_INPUT PERSISTENT
	{attribute 'OPC.UA.DA' := '1'}
	SP AT %M* :  REAL:=100;	//Börvärde~wp:[unit]Pa[format]0
	{attribute 'OPC.UA.DA' := '1'}
	ESP AT %M* : REAL:=0; //Externt börvärde (Absolutbörvärde)~wp:[unit]Pa[format]0
END_VAR

VAR_OUTPUT
	{attribute 'OPC.UA.DA' := '1'}
	CSP AT %M*: REAL; //Uträknat börvärde~wp:[unit]Pa[format]0
	{attribute 'OPC.UA.DA' := '1'}
	ISP AT %M* : REAL:=0; //Börvärde från optimering~wp:[unit]Pa[format]0
		
END_VAR

	SUPER^(); 
	//Börvärde
	rSetpoint := SP;
	
	//Läs från bas	
	CSP := rCSP;
	ISP := rIspInternal;
	//Skriv till bas
	rMin := MIN(ISP, SP, ESP) + rPowerLimitOffset;
	rMax := MAX(ISP,SP, ESP) + rPowerLimitOffset;
	rESP := ESP;
	bSetpointTypeBase := 'Internt börvärde';

END_FUNCTION_BLOCK

// oaksLibrary/Börvärden/SetPointOutdoorCompCDewpoint
FUNCTION_BLOCK SetPointOutdoorCompCDewpoint EXTENDS fbSetPointOutdoorCompC
VAR_INPUT
	rDewpointTemperature : REAL; 
	rDewpointHumidity : REAL;
END_VAR	
VAR
	fbDewpointCalc01 : fbDewpointCalc;
END_VAR
VAR_OUTPUT
	rCalculatedDewpoint : REAL; // Uträknad daggpunkt
END_VAR
VAR_IN_OUT
	rSetpointAdjust : REAL; //Börvärdesförskjutning över uträknad daggpunkt
END_VAR

	SUPER^(); 
	bAktiveraSkrivningCsp := FALSE; // Inaktivera skrivning i basblock för att kunna skriva csp från detta block.

	IF rSetpointAdjust < 0.5 THEN
		rSetpointAdjust := 0.5;
	END_IF

	SUPER^(); 
	
	fbDewpointCalc01(
	rTemperature:= rDewpointTemperature, 
	rRelativeHumidity:= rDewpointHumidity, 
	rSetpointOffest:=rSetpointAdjust , 
	rSetpoint:=rCSP,
	PV=> rCalculatedDewpoint, 
	rCSP=> );

	//Skriv till bas	
	CSP := fbDewpointCalc01.rCSP;

END_FUNCTION_BLOCK

// oaksLibrary/Datahantering/F_GetTempToUseMeanTemp
//Funktion för att välja vilken utetemperatur som ska användas. Knyter man ingenting väljs  oaksGVL.rOutdoorTempMean. Knyter man en REAL väljs det värdet.
FUNCTION F_GetTempToUseMeanTemp : REAL
VAR_INPUT
	rTempToUse : ANY; //Temperatur för start/stopp. Om inget kopplas används oaksGVL.rOutdoorTempMean
END_VAR
VAR
	pAnyReal : POINTER TO REAL;
END_VAR

//Temp select
IF rTempToUse.TypeClass = __SYSTEM.TYPE_CLASS.TYPE_REAL THEN
	pAnyReal := rTempToUse.pValue;
	F_GetTempToUseMeanTemp := pAnyReal^;
ELSE
	F_GetTempToUseMeanTemp := oaksGVL.rOutdoorTempMean;
END_IF

END_FUNCTION

// oaksLibrary/Datahantering/FbDoubleControlledVariable
FUNCTION_BLOCK FbDoubleControlledVariable
VAR_IN_OUT
	nVariableInPLC			:	INT;
	nVariableInModbusUnit	:	INT;
END_VAR
VAR_OUTPUT
END_VAR
VAR
	nSavedData				:	INT;
END_VAR

IF nVariableInModbusUnit <> nSavedData THEN
	nVariableInPLC:=nVariableInModbusUnit;
	nSavedData:=nVariableInModbusUnit;
ELSIF nVariableInPLC <> nSavedData THEN
	nVariableInModbusUnit:=nVariableInPLC;
	nSavedData:=nVariableInPLC;
END_IF

END_FUNCTION_BLOCK

// oaksLibrary/Datahantering/FbDoubleControlledVariableLreal
FUNCTION_BLOCK FbDoubleControlledVariableLreal
VAR_IN_OUT
	lRVariableInPLC			:	LREAL;
	lRVariableInModbusUnit	:	LREAL;
END_VAR
VAR_OUTPUT
END_VAR
VAR
	lRSavedData				:	LREAL;
END_VAR

IF lRVariableInModbusUnit <> lRSavedData THEN
	lRVariableInPLC:=lRVariableInModbusUnit;
	lRSavedData:=lRVariableInModbusUnit;
ELSIF lRVariableInPLC <> lRSavedData THEN
	lRVariableInModbusUnit:=lRVariableInPLC;
	lRSavedData:=lRVariableInPLC;
END_IF

END_FUNCTION_BLOCK

// oaksLibrary/Datahantering/FbDoubleControlledVariableReal
FUNCTION_BLOCK FbDoubleControlledVariableReal
VAR_IN_OUT
	rVariableInPLC			:	REAL;
	rVariableInModbusUnit	:	REAL;
END_VAR
VAR_OUTPUT
END_VAR
VAR
	rSavedData				:	REAL;
END_VAR

IF rVariableInModbusUnit <> rSavedData THEN
	rVariableInPLC:=rVariableInModbusUnit;
	rSavedData:=rVariableInModbusUnit;
ELSIF rVariableInPLC <> rSavedData THEN
	rVariableInModbusUnit:=rVariableInPLC;
	rSavedData:=rVariableInPLC;
END_IF

END_FUNCTION_BLOCK

// oaksLibrary/Datahantering/FbDoubleControlledVariableRealToWord
FUNCTION_BLOCK FbDoubleControlledVariableRealToWord
VAR_INPUT
	rScale : REAL := 10;
END_VAR
VAR_IN_OUT
	rVariableInPLC			:	REAL;
	wVariableInModbusUnit	:	WORD;
END_VAR
VAR_OUTPUT
END_VAR
VAR
	rSavedData				:	REAL;
	dIntTemp : DINT;
	rTemp : REAL;
END_VAR

IF wVariableInModbusUnit <> (rSavedData * rScale) THEN
	rTemp := wVariableInModbusUnit;
	rVariableInPLC:=rTemp / rScale;
	rSavedData:=rTemp / rScale;
ELSIF rVariableInPLC <> rSavedData THEN
	rTemp := rVariableInPLC  * rScale;
	dIntTemp := REAL_TO_DINT(rTemp);
	wVariableInModbusUnit:=DINT_TO_WORD(dIntTemp);
	rSavedData:=rVariableInPLC;
END_IF

END_FUNCTION_BLOCK

// oaksLibrary/Datahantering/FbDoubleControlledVariableWord
FUNCTION_BLOCK FbDoubleControlledVariableWord
VAR_IN_OUT
	wVariableInPLC			:	WORD;
	wVariableInModbusUnit	:	WORD;
END_VAR
VAR_OUTPUT
END_VAR
VAR
	wSavedData				:	WORD;
END_VAR

IF wVariableInModbusUnit <> wSavedData THEN
	wVariableInPLC:=wVariableInModbusUnit;
	wSavedData:=wVariableInModbusUnit;
ELSIF wVariableInPLC <> wSavedData THEN
	wVariableInModbusUnit:=wVariableInPLC;
	wSavedData:=wVariableInPLC;
END_IF

END_FUNCTION_BLOCK

// oaksLibrary/Datahantering/fbModbusSekvensArray
FUNCTION_BLOCK fbModbusSekvensArray
VAR_INPUT
	
END_VAR
VAR_OUTPUT
	{attribute 'OPC.UA.DA' := '1'}
	PV AT %M* 	: INT; //Aktuell modbus-id loop 1~wp:
	{attribute 'OPC.UA.DA' := '1'}
	PV1 AT %M* : INT; //Aktuell modbus-id loop 2~wp:
	{attribute 'OPC.UA.DA' := '1'}
	PV2 AT %M*  : INT; //Aktuell modbus-id loop 3~wp:
	{attribute 'OPC.UA.DA' := '1'}
	PV3 AT %M*  : INT; //Aktuell modbus-id loop 4~wp:
	{attribute 'OPC.UA.DA' := '1'}
	PV4 AT %M*  : INT; //Aktuell modbus-id loop 5~wp:
	{attribute 'OPC.UA.DA' := '1'}
	PV5 AT %M*  : INT; //Aktuell modbus-id loop 6~wp:
	{attribute 'OPC.UA.DA' := '1'}
	PV6 AT %M*  : INT; //Aktuell modbus-id loop 7~wp:
	{attribute 'OPC.UA.DA' := '1'}
	PV7 AT %M*  : INT; //Aktuell modbus-id loop 8~wp:
	{attribute 'OPC.UA.DA' := '1'}
	PV8 AT %M*  : INT; //Aktuell modbus-id loop 9~wp:
	{attribute 'OPC.UA.DA' := '1'}
	PV9 AT %M*  : INT; //Aktuell modbus-id loop 10~wp:
	{attribute 'OPC.UA.DA' := '1'}
	PV10 AT %M*  : INT; //Aktuell modbus-id loop 11~wp:
	{attribute 'OPC.UA.DA' := '1'}
	PV11 AT %M*  : INT; //Aktuell modbus-id loop 12~wp:
	{attribute 'OPC.UA.DA' := '1'}
	PV12 AT %M*  : INT; //Aktuell modbus-id loop 13~wp:
	{attribute 'OPC.UA.DA' := '1'}
	PV13 AT %M*  : INT; //Aktuell modbus-id loop 14~wp:
	{attribute 'OPC.UA.DA' := '1'}
	PV14 AT %M*  : INT; //Aktuell modbus-id loop 15~wp:				
	{attribute 'OPC.UA.DA' := '1'}
	PV15 AT %M*  : INT; //Aktuell modbusadress loop 16~wp:	
END_VAR
VAR
	{attribute 'OPC.UA.DA' := '1'}
	SEKVENS1_PV 	AT %M* : INT; //Aktuell modbus-id loop 1~wp:
	{attribute 'OPC.UA.DA' := '1'}
	SEKVENS2_PV 	AT %M* : INT; //Aktuell modbus-id loop 2~wp:
	{attribute 'OPC.UA.DA' := '1'}
	SEKVENS3_PV 	AT %M* : INT; //Aktuell modbus-id loop 3~wp:
	{attribute 'OPC.UA.DA' := '1'}
	SEKVENS4_PV 	AT %M* : INT; //Aktuell modbus-id loop 4~wp:
	{attribute 'OPC.UA.DA' := '1'}
	SEKVENS5_PV 	AT %M* : INT; //Aktuell modbus-id loop 5~wp:
	{attribute 'OPC.UA.DA' := '1'}
	SEKVENS6_PV 	AT %M* : INT; //Aktuell modbus-id loop 6~wp:
	{attribute 'OPC.UA.DA' := '1'}
	SEKVENS7_PV 	AT %M* : INT; //Aktuell modbus-id loop 7~wp:
	{attribute 'OPC.UA.DA' := '1'}
	SEKVENS8_PV 	AT %M* : INT; //Aktuell modbus-id loop 8~wp:
	{attribute 'OPC.UA.DA' := '1'}
	SEKVENS9_PV 	AT %M* : INT; //Aktuell modbus-id loop 9~wp:
	{attribute 'OPC.UA.DA' := '1'}
	SEKVENS10_PV 	AT %M* : INT; //Aktuell modbus-id loop 10~wp:
	{attribute 'OPC.UA.DA' := '1'}
	SEKVENS11_PV 	AT %M* : INT; //Aktuell modbus-id loop 11~wp:
	{attribute 'OPC.UA.DA' := '1'}
	SEKVENS12_PV 	AT %M* : INT; //Aktuell modbus-id loop 12~wp:
	{attribute 'OPC.UA.DA' := '1'}
	SEKVENS13_PV 	AT %M* : INT; //Aktuell modbus-id loop 13~wp:
	{attribute 'OPC.UA.DA' := '1'}
	SEKVENS14_PV 	AT %M* : INT; //Aktuell modbus-id loop 14~wp:
	{attribute 'OPC.UA.DA' := '1'}
	SEKVENS15_PV 	AT %M* : INT; //Aktuell modbus-id loop 15~wp:
	{attribute 'OPC.UA.DA' := '1'}
	SEKVENS16_PV 	AT %M* : INT; //Aktuell modbusadress loop 16~wp:
	
	iTemp : INT; // används för temporär lagring	

	TON01sekvens1 : TON;
	TON02sekvens1 : TON;
		
	TON01sekvens2 : TON;
	TON02sekvens2 : TON;
		
	TON01sekvens3 : TON;
	TON02sekvens3 : TON;
		
	TON01sekvens4 : TON;
	TON02sekvens4 : TON;
		
	TON01sekvens5 : TON;
	TON02sekvens5 : TON;
		
	TON01sekvens6 : TON;
	TON02sekvens6 : TON;
		
	TON01sekvens7 : TON;
	TON02sekvens7 : TON;
		
	TON01sekvens8 : TON;
	TON02sekvens8 : TON;
		
	TON01sekvens9 : TON;
	TON02sekvens9 : TON;
		
	TON01sekvens10 : TON;
	TON02sekvens10 : TON;
	
	TON01sekvens11 : TON;
	TON02sekvens11 : TON;
	
	TON01sekvens12 : TON;
	TON02sekvens12 : TON;
	
	TON01sekvens13 : TON;
	TON02sekvens13 : TON;
	
	TON01sekvens14 : TON;
	TON02sekvens14 : TON;
	
	TON01sekvens15 : TON;
	TON02sekvens15 : TON;
	
	TON01sekvens16 : TON; // Denna används för exempelvis elvaco då man har många läsningar mot en enhet
	TON02sekvens16 : TON; // Denna används för exempelvis elvaco då man har många läsningar mot en enhet
		
END_VAR
VAR_INPUT PERSISTENT
	SekvensLasFordrojning1 : TIME := T#1S;	//Läsfördröjning
	SekvensTimeouttid1 : TIME := T#5S;		//Timeouttid 
	SekvensMinID1 : INT := 1;				//Första adress på slingan
	SekvensMaxID1 : INT := 253;				//Sista adress på slingan
	
	SekvensLasFordrojning2 : TIME := T#1S;
	SekvensTimeouttid2 : TIME := T#5S;
	SekvensMinID2 : INT := 1;				
	SekvensMaxID2 : INT := 253;				
	
	SekvensLasFordrojning3 : TIME := T#1S;
	SekvensTimeouttid3 : TIME := T#5S;
	SekvensMinID3 : INT := 1;				
	SekvensMaxID3 : INT := 253;				
	
	SekvensLasFordrojning4 : TIME := T#1S;
	SekvensTimeouttid4 : TIME := T#5S;
	SekvensMinID4 : INT := 1;				
	SekvensMaxID4 : INT := 253;				
	
	SekvensLasFordrojning5 : TIME := T#1S;
	SekvensTimeouttid5 : TIME := T#5S;
	SekvensMinID5 : INT := 1;				
	SekvensMaxID5 : INT := 253;				
	
	SekvensLasFordrojning6 : TIME := T#1S;
	SekvensTimeouttid6 : TIME := T#5S;
	SekvensMinID6 : INT := 1;				
	SekvensMaxID6 : INT := 253;		
	
	SekvensLasFordrojning7 : TIME := T#1S;
	SekvensTimeouttid7 : TIME := T#5S;
	SekvensMinID7 : INT := 1;				
	SekvensMaxID7 : INT := 253;		
	
	SekvensLasFordrojning8 : TIME := T#1S;
	SekvensTimeouttid8 : TIME := T#5S;
	SekvensMinID8 : INT := 1;				
	SekvensMaxID8 : INT := 253;		
	
	SekvensLasFordrojning9 : TIME := T#1S;
	SekvensTimeouttid9 : TIME := T#5S;
	SekvensMinID9 : INT := 1;				
	SekvensMaxID9 : INT := 253;		
	
	SekvensLasFordrojning10 : TIME := T#1S;
	SekvensTimeouttid10 : TIME := T#5S;
	SekvensMinID10 : INT := 1;				
	SekvensMaxID10 : INT := 253;		
	
	SekvensLasFordrojning11 : TIME := T#1S;
	SekvensTimeouttid11 : TIME := T#5S;
	SekvensMinID11 : INT := 1;				
	SekvensMaxID11 : INT := 253;		
	
	SekvensLasFordrojning12 : TIME := T#1S;
	SekvensTimeouttid12 : TIME := T#5S;
	SekvensMinID12 : INT := 1;				
	SekvensMaxID12 : INT := 253;		
	
	SekvensLasFordrojning13 : TIME := T#1S;
	SekvensTimeouttid13 : TIME := T#5S;
	SekvensMinID13 : INT := 1;				
	SekvensMaxID13 : INT := 253;		
	
	SekvensLasFordrojning14 : TIME := T#1S;
	SekvensTimeouttid14 : TIME := T#5S;
	SekvensMinID14 : INT := 1;				
	SekvensMaxID14 : INT := 253;		
	
	SekvensLasFordrojning15 : TIME := T#1S;
	SekvensTimeouttid15 : TIME := T#5S;
	SekvensMinID15 : INT := 1;				
	SekvensMaxID15 : INT := 253;		
	
	SekvensLasFordrojning16 : TIME := T#1S; // Denna används för exempelvis elvaco då man har många läsningar mot en enhet
	SekvensTimeouttid16 : TIME := T#5S; // Denna används för exempelvis elvaco då man har många läsningar mot en enhet
	//SekvensMinID16 : INT := 1;	
	//SekvensMaxID16 : INT := 253;		
END_VAR


mModbusSekvens(TON01sekvens1,TON02sekvens1,1,oaksGVL.bEnableSekvens1,SekvensLasFordrojning1,SekvensTimeouttid1, SekvensMinID1, SekvensMaxID1, PV=>PV, SEKVENS_PV=>SEKVENS1_PV);
mModbusSekvens(TON01sekvens2,TON02sekvens2,2,oaksGVL.bEnableSekvens2,SekvensLasFordrojning2,SekvensTimeouttid2, SekvensMinID2, SekvensMaxID2, PV=>PV1, SEKVENS_PV=>SEKVENS2_PV);
mModbusSekvens(TON01sekvens3,TON02sekvens3,3,oaksGVL.bEnableSekvens3,SekvensLasFordrojning3,SekvensTimeouttid3, SekvensMinID3, SekvensMaxID3, PV=>PV2, SEKVENS_PV=>SEKVENS3_PV);
mModbusSekvens(TON01sekvens4,TON02sekvens4,4,oaksGVL.bEnableSekvens4,SekvensLasFordrojning4,SekvensTimeouttid4, SekvensMinID4, SekvensMaxID4, PV=>PV3, SEKVENS_PV=>SEKVENS4_PV);
mModbusSekvens(TON01sekvens5,TON02sekvens5,5,oaksGVL.bEnableSekvens5,SekvensLasFordrojning5,SekvensTimeouttid5, SekvensMinID5, SekvensMaxID5, PV=>PV4, SEKVENS_PV=>SEKVENS5_PV);
mModbusSekvens(TON01sekvens6,TON02sekvens6,6,oaksGVL.bEnableSekvens6,SekvensLasFordrojning6,SekvensTimeouttid6, SekvensMinID6, SekvensMaxID6, PV=>PV5, SEKVENS_PV=>SEKVENS6_PV);
mModbusSekvens(TON01sekvens7,TON02sekvens7,7,oaksGVL.bEnableSekvens7,SekvensLasFordrojning7,SekvensTimeouttid7, SekvensMinID7, SekvensMaxID7, PV=>PV6, SEKVENS_PV=>SEKVENS7_PV);
mModbusSekvens(TON01sekvens8,TON02sekvens8,8,oaksGVL.bEnableSekvens8,SekvensLasFordrojning8,SekvensTimeouttid8, SekvensMinID8, SekvensMaxID8, PV=>PV7, SEKVENS_PV=>SEKVENS8_PV);
mModbusSekvens(TON01sekvens9,TON02sekvens9,9,oaksGVL.bEnableSekvens9,SekvensLasFordrojning9,SekvensTimeouttid9 ,SekvensMinID9,  SekvensMaxID9, PV=>PV8, SEKVENS_PV=>SEKVENS9_PV);
mModbusSekvens(TON01sekvens10,TON02sekvens10,10,oaksGVL.bEnableSekvens10,SekvensLasFordrojning10,SekvensTimeouttid10, SekvensMinID10, SekvensMaxID10, PV=>PV9, SEKVENS_PV=>SEKVENS10_PV);
mModbusSekvens(TON01sekvens11,TON02sekvens11,11,oaksGVL.bEnableSekvens11,SekvensLasFordrojning11,SekvensTimeouttid11, SekvensMinID11, SekvensMaxID11, PV=>PV10, SEKVENS_PV=>SEKVENS11_PV);
mModbusSekvens(TON01sekvens12,TON02sekvens12,12,oaksGVL.bEnableSekvens12,SekvensLasFordrojning12,SekvensTimeouttid12, SekvensMinID12, SekvensMaxID12, PV=>PV11, SEKVENS_PV=>SEKVENS12_PV);
mModbusSekvens(TON01sekvens13,TON02sekvens13,13,oaksGVL.bEnableSekvens13,SekvensLasFordrojning13,SekvensTimeouttid13, SekvensMinID13, SekvensMaxID13, PV=>PV12, SEKVENS_PV=>SEKVENS13_PV);
mModbusSekvens(TON01sekvens14,TON02sekvens14,14,oaksGVL.bEnableSekvens14,SekvensLasFordrojning14,SekvensTimeouttid14, SekvensMinID14, SekvensMaxID14, PV=>PV13, SEKVENS_PV=>SEKVENS14_PV);
mModbusSekvens(TON01sekvens15,TON02sekvens15,15,oaksGVL.bEnableSekvens15,SekvensLasFordrojning15,SekvensTimeouttid15, SekvensMinID15, SekvensMaxID15, PV=>PV14, SEKVENS_PV=>SEKVENS15_PV);


// Denna används för exempelvis elvaco då man har många läsningar mot en enhet
mModbusSekvensUppTill1000(TON01sekvens16,TON02sekvens16,16,oaksGVL.bEnableSekvens16,SekvensLasFordrojning16,SekvensTimeouttid16, PV=>PV15, SEKVENS_PV=>SEKVENS16_PV);

METHOD PRIVATE mModbusSekvens
VAR_IN_OUT
	TON01 : TON;
	TON02 : TON;
END_VAR
VAR_INPUT
	iSekvens : INT;
	bEnableSekvens : BOOL;
	tLasFordrojning : TIME;
	tTimeouttid : TIME;
	iMinID	: INT;
	iMaxID	: INT;
END_VAR
VAR_OUTPUT
	PV : INT;
	SEKVENS_PV 		: INT;
END_VAR
(* Kommer funktion för handställning vid senare tillfälle *)
	IF iMaxID > 255 THEN iMaxID := 255; END_IF;
	IF iMinID > iMaxID THEN iMinID := iMaxID; END_IF;

	IF (NOT oaksgvl.aBModbusBusyFlagga[iSekvens,oaksgvl.aBModbusSekvens[iSekvens]] OR TON02.Q) AND bEnableSekvens THEN
		TON01(IN:=TRUE , PT:=tLasFordrojning , Q=> , ET=> );
		TON02(IN:=FALSE , PT:=tTimeouttid , Q=> , ET=> );	
		IF TON01.Q THEN
			iTemp := MAX(iMinID, oaksgvl.aBModbusSekvens[iSekvens]);
			oaksgvl.aBModbusSekvens[iSekvens] := iTemp + 1;
			IF oaksgvl.aBModbusSekvens[iSekvens] > iMaxID THEN
				oaksgvl.aBModbusSekvens[iSekvens] := iMinID;
			END_IF
		END_IF
	ELSE
		TON01(IN:=FALSE , PT:=tLasFordrojning , Q=> , ET=> );	
		TON02(IN:=TRUE , PT:=tTimeouttid , Q=> , ET=> );	
	END_IF

PV := oaksgvl.aBModbusSekvens[iSekvens];
SEKVENS_PV := oaksgvl.aBModbusSekvens[iSekvens];
END_METHOD

METHOD mModbusSekvensUppTill1000
VAR_IN_OUT
	TON01 : TON;
	TON02 : TON;
END_VAR
VAR_INPUT
	iSekvens : INT;
	bEnableSekvens : BOOL;
	tLasFordrojning : TIME;
	tTimeouttid : TIME;
END_VAR
VAR_OUTPUT
	PV : INT;
	SEKVENS_PV 		: INT;
END_VAR
(* Kommer funktion för handställning vid senare tillfälle *)
	IF (NOT oaksgvl.aBModbusBusyFlaggaAdresser[iSekvens-15,oaksgvl.aBModbusSekvens[iSekvens]] OR TON02.Q) AND bEnableSekvens THEN
		TON01(IN:=TRUE , PT:=tLasFordrojning , Q=> , ET=> );
		TON02(IN:=FALSE , PT:=tTimeouttid , Q=> , ET=> );	
		IF TON01.Q THEN
			iTemp := oaksgvl.aBModbusSekvens[iSekvens];
			oaksgvl.aBModbusSekvens[iSekvens] := iTemp + 1;
			IF oaksgvl.aBModbusSekvens[iSekvens] = 2998  THEN
				oaksgvl.aBModbusSekvens[iSekvens] := 1;
			END_IF
		END_IF
	ELSE
		TON01(IN:=FALSE , PT:=tLasFordrojning , Q=> , ET=> );	
		TON02(IN:=TRUE , PT:=tTimeouttid , Q=> , ET=> );	
	END_IF

PV := oaksgvl.aBModbusSekvens[iSekvens];
SEKVENS_PV := oaksgvl.aBModbusSekvens[iSekvens];
END_METHOD

END_FUNCTION_BLOCK

// oaksLibrary/Datahantering/fDwordToWordHigh
// slår ihop två 16 bitars tal till ett 32 bitars tal. Exempelvis för att slå ihop två modbusregister.
FUNCTION fDwordToWordHigh : WORD
VAR_INPUT
	wInput : DWORD;
END_VAR
VAR
END_VAR

	fDwordToWordHigh.0  := wInput.16; 
	fDwordToWordHigh.1  := wInput.17; 
	fDwordToWordHigh.2  := wInput.18; 
	fDwordToWordHigh.3  := wInput.19; 
	fDwordToWordHigh.4  := wInput.20; 
	fDwordToWordHigh.5  := wInput.21; 
	fDwordToWordHigh.6  := wInput.22; 
	fDwordToWordHigh.7  := wInput.23; 
	fDwordToWordHigh.8  := wInput.24; 
	fDwordToWordHigh.9  := wInput.25; 
	fDwordToWordHigh.10 := wInput.26;
	fDwordToWordHigh.11 := wInput.27;
	fDwordToWordHigh.12 := wInput.28;
	fDwordToWordHigh.13 := wInput.29;
	fDwordToWordHigh.14 := wInput.30;
	fDwordToWordHigh.15 := wInput.31;

END_FUNCTION

// oaksLibrary/Datahantering/fDwordToWordLow
// slår ihop två 16 bitars tal till ett 32 bitars tal. Exempelvis för att slå ihop två modbusregister.
FUNCTION fDwordToWordLow : WORD
VAR_INPUT
	wInput : DWORD;
END_VAR
VAR
END_VAR

	fDwordToWordLow.0  := wInput.0; 
	fDwordToWordLow.1  := wInput.1; 
	fDwordToWordLow.2  := wInput.2; 
	fDwordToWordLow.3  := wInput.3; 
	fDwordToWordLow.4  := wInput.4; 
	fDwordToWordLow.5  := wInput.5; 
	fDwordToWordLow.6  := wInput.6; 
	fDwordToWordLow.7  := wInput.7; 
	fDwordToWordLow.8  := wInput.8; 
	fDwordToWordLow.9  := wInput.9; 
	fDwordToWordLow.10 := wInput.10;
	fDwordToWordLow.11 := wInput.11;
	fDwordToWordLow.12 := wInput.12;
	fDwordToWordLow.13 := wInput.13;
	fDwordToWordLow.14 := wInput.14;
	fDwordToWordLow.15 := wInput.15;

END_FUNCTION

// oaksLibrary/Datahantering/fRealToWord
// Använd denna vid konvertering från real till word. Hanterar även negativa tal. Använd alltid denna istället för REAL_TO_WORD
FUNCTION fRealToWord : WORD
VAR_INPUT
	rReal : REAL;
	uiFaktor : REAL;
END_VAR
VAR
	rTemp  :REAL;
	dint1 : dint;
END_VAR

rTemp := rReal *uiFaktor;

dint1 := REAL_TO_DINT(rTemp);

fRealToWord := DINT_TO_WORD(dint1);

END_FUNCTION

// oaksLibrary/Datahantering/fSetpointLimiter
//Oaks AB
//2022-06-07
///Funktion för att begränsa ett inställt värde mellan min-/maxbegränsning.
FUNCTION fSetpointLimiter : REAL
VAR_INPUT
	rMin : REAL :=0;
	rMax : REAL :=0;
END_VAR
VAR
END_VAR
VAR_IN_OUT
	rValue : REAL; 
END_VAR

IF rValue >= rMax THEN
	rValue := rMax;
ELSIF rValue <= rMin THEN
	rValue := rMin;
END_IF

fSetpointLimiter := rValue;

END_FUNCTION

// oaksLibrary/Datahantering/fSignedConverter
// signed konvertering 16 bits tal. Går talet över 32767 indikeras negativt tal.
FUNCTION fSignedConverter : REAL
VAR_INPUT
	rInput : REAL;
END_VAR
VAR
	iTemp : INT;
END_VAR

	IF rInput > 32767 THEN
		fSignedConverter := (rInput - 65536); 
	ELSE
		fSignedConverter := rInput;
	END_IF

END_FUNCTION

// oaksLibrary/Datahantering/fSignedDoubleConverter
// signed konvertering 32 bits tal. Går talet över 2147483647 indikeras negativt tal.
FUNCTION fSignedDoubleConverter : REAL
VAR_INPUT
	rInput : REAL;
END_VAR
VAR
END_VAR


	IF rInput > 2147483647 THEN
		fSignedDoubleConverter :=  (rInput - 4294967296) / 100;
	ELSE
		fSignedDoubleConverter := rInput / 100;
	END_IF

END_FUNCTION

// oaksLibrary/Datahantering/fWordToDoubleWord
// slår ihop två 16 bitars tal till ett 32 bitars tal. Exempelvis för att slå ihop två modbusregister.
FUNCTION fWordToDoubleWord : DWORD
VAR_INPUT
	wInput1 : WORD;
	wInput2 : WORD;
END_VAR
VAR
END_VAR

	fWordToDoubleWord.0  := wInput1.0; 
	fWordToDoubleWord.1  := wInput1.1; 
	fWordToDoubleWord.2  := wInput1.2; 
	fWordToDoubleWord.3  := wInput1.3; 
	fWordToDoubleWord.4  := wInput1.4; 
	fWordToDoubleWord.5  := wInput1.5; 
	fWordToDoubleWord.6  := wInput1.6; 
	fWordToDoubleWord.7  := wInput1.7; 
	fWordToDoubleWord.8  := wInput1.8; 
	fWordToDoubleWord.9  := wInput1.9; 
	fWordToDoubleWord.10 := wInput1.10;
	fWordToDoubleWord.11 := wInput1.11;
	fWordToDoubleWord.12 := wInput1.12;
	fWordToDoubleWord.13 := wInput1.13;
	fWordToDoubleWord.14 := wInput1.14;
	fWordToDoubleWord.15 := wInput1.15;
																		   
	fWordToDoubleWord.16 :=wInput2.0; 
	fWordToDoubleWord.17 :=wInput2.1; 
	fWordToDoubleWord.18 :=wInput2.2; 
	fWordToDoubleWord.19 :=wInput2.3; 
	fWordToDoubleWord.20 :=wInput2.4; 
	fWordToDoubleWord.21 :=wInput2.5; 
	fWordToDoubleWord.22 :=wInput2.6; 
	fWordToDoubleWord.23 :=wInput2.7; 
	fWordToDoubleWord.24 :=wInput2.8; 
	fWordToDoubleWord.25 :=wInput2.9; 
	fWordToDoubleWord.26 :=wInput2.10; 
	fWordToDoubleWord.27 :=wInput2.11; 
	fWordToDoubleWord.28 :=wInput2.12; 
	fWordToDoubleWord.29 :=wInput2.13; 
	fWordToDoubleWord.30 :=wInput2.14; 
	fWordToDoubleWord.31 :=wInput2.15;

END_FUNCTION

// oaksLibrary/EtherCAT Specifikt/Givare/fbOutDoorTempMeanEL3204
FUNCTION_BLOCK fbOutDoorTempMeanEL3204 EXTENDS fbPtEL3204
VAR_OUTPUT
	{attribute 'OPC.UA.DA' := '1'}
	PV1 AT %M*  : REAL; //Medeltemperatur~wp:[unit]°C[format]0.0[trendoptions]i:300
END_VAR
VAR
	bResetMeanTemp : BOOL; //Sätt denna till TRUE för återställning av medelvärdesberäkning.
	lrMeanInternal : LREAL;
	lrMeanInternalTemp : LREAL;
//	fbPLC_SystemTime: Tc3_BA.FB_BA_GetTime;
	stTime		: tc2_ba.TIMESTRUCT;

	FB_BA_GetTime01 : tc2_ba.FB_BA_GetTime; 
//	FB_BA_ExtTiSt01 : tc2_ba.FB_BA_ExtTiSt;	

//	wMinute : WORD;
	fbMinuteTrig : R_TRIG;
	//iTemp : INT;
	iCounter : UINT := 4319;
	
	iAntalMinuterMedel : UINT;
	iAntalMinuterForUtrakning : UINT; //Maxbegränsar antal minuter som används för beräkning beroende på hur många minuter som finns insamlade
END_VAR
VAR PERSISTENT
	wLastMinuteOfChange : WORD;	
	{attribute 'OPC.UA.DA' := '1'}
	PV7 AT %M* : UINT;  //Antal minuter insamlade för medelvärdesberäkning (max 4320)~wp:[unit]minuter[format]0

	rArrayMean72Hours : ARRAY [0..4319] OF REAL;
END_VAR
VAR_INPUT PERSISTENT
	{attribute 'OPC.UA.DA' := '1'}
	SP1 AT %M* : UINT := 12; //Antal timmar för medelvärdesberäkning (2-72)~wp:[unit]timmar[format]0
END_VAR

	SUPER^();

	IF bResetMeanTemp THEN
		bResetMeanTemp := FALSE;
		PV7 := 2;
	END_IF

	IF SP1 > 72 THEN // Medelvärdestid maxbegränsas till 72 timmar.
		SP1 := 72;
	ELSIF SP1 < 2 THEN // Medelvärdestid minbegränsas till 2 timmar.
		SP1 := 2;
	END_IF
	
	IF SP1 <= 72 AND SP1 > 1 THEN
		 iAntalMinuterMedel := SP1 * 60;
	END_IF;


	mMean(); // Metod för att räkna ut medelvärde
	//4320 minuter = 72 timmar.
	IF iAntalMinuterForUtrakning > 2 THEN
		PV1 := LREAL_TO_REAL(lrMeanInternal) / iAntalMinuterForUtrakning; 
	END_IF;
	
	//oaksGVL.rOutdoorTemp := mPv(TRUE); //utetemp som behåller sitt senaste giltiga värde vid givarfel 
	
	oaksGVL.rOutdoorTemp := PV;	//Utetemp som behåller sitt senaste giltliga värde vid givarfel, alternativ att sätta inställbart värde
	
	IF NOT FAULT THEN 
		oaksGVL.rOutdoorTempErrorValue0 := PV; // global utetemp som ställs till 0 vid givarfel.
		oaksGVL.rOutdoorTempErrorValue150 := PV;// global utetemp som ställs till 150 vid givarfel.
	ELSE
		oaksGVL.rOutdoorTempErrorValue0 := 0; // global utetemp som ställs till 0 vid givarfel.
		oaksGVL.rOutdoorTempErrorValue150 := 150;// global utetemp som ställs till 150 vid givarfel.
	END_IF
	oaksGVL.rOutdoorTempMean := PV1; // global medel utetemp
	
	oaksGVL.bOutdoorTempSensorError := FAULT; // globalt utegivarfel

METHOD PRIVATE mMean : BOOL
VAR_INPUT
END_VAR
	FB_BA_GetTime01(bEn :=TRUE);	
	stTime := FB_BA_GetTime01.stSysTi;

	IF stTime.wMinute <> wLastMinuteOfChange THEN
		fbMinuteTrig(CLK := TRUE);
	ELSE
		fbMinuteTrig(CLK := FALSE);
	END_IF
	//4320 minuter - 1 = 72 timmar.
	IF fbMinuteTrig.Q THEN
		FOR iCounter:= iAntalMinuterMedel - 1 TO 1 BY -1 DO
			rArrayMean72Hours[iCounter]:=rArrayMean72Hours[iCounter-1];
		END_FOR;
		rArrayMean72Hours[0] := PV;
		wLastMinuteOfChange := stTime.wMinute;
		IF PV7 < 4320 THEN // Räknas upp för att hålla koll på antal insamlade minuter
			PV7 := PV7 +1;
		END_IF
	END_IF 
	
	lrMeanInternal := 0;
	//4320 minuter - 1 = 72 timmar.
	iAntalMinuterForUtrakning := MIN(iAntalMinuterMedel,PV7); // Max begränsar antal minuter som används för beräkning beroende på hur många minuter som finns insamlade
	FOR iCounter:= iAntalMinuterForUtrakning TO 1 BY -1 DO
		lrMeanInternalTemp := lrMeanInternal;
		lrMeanInternal:=rArrayMean72Hours[iCounter-1] + lrMeanInternalTemp;
	END_FOR;
END_METHOD

END_FUNCTION_BLOCK

// oaksLibrary/EtherCAT Specifikt/Givare/fbPtEL3204
FUNCTION_BLOCK fbPtEL3204
VAR_INPUT
	{attribute 'OPC.UA.DA' := '1'}
	M AT %M* : BOOL;//Handställning~wp:[trendoptions]i:14400, t:1
	bFaultVal : BOOL := FALSE; //TRUE = Behåller senaste värde vid givarfel, FALSE = 150 vid kabelbrott, 0 vid kortslutning
	rFaultVal : REAL:=-999; //Om bFaultVal är TRUE så kan man välja temperatur som skall hållas här. Väljer man inget tar den senaste värdet givaren hade innan givarfel
	//OBS Tar man bort funtkion för rFaultVal i efterhand men vill behålla senaste värde (bFaultVal = TRUE) behöver man sätta rFaultVal till -999
END_VAR
VAR_OUTPUT
	{attribute 'OPC.UA.DA' := '1'}
	PV AT %M* : REAL;//Temperatur~wp:[unit]°C[format]0.0[trendoptions]i:300
	{attribute 'OPC.UA.DA' := '1'}
	FAULT AT %M* : BOOL;//Givarfel~wp:
	{attribute 'OPC.UA.DA' := '1'}
	AL8 AT %M* : BOOL; //Givare handställd~wp:[alarmoptions]p:3:
END_VAR
VAR
	fbAlarm2, fbAlarm1 : fbAlarm; // Larm handställning
	iDataIn AT %I*: INT;
	FB_BA_TiAvrg01,FB_BA_TiAvrg02 : tc2_ba.FB_BA_TiAvrg;
END_VAR
VAR_INPUT PERSISTENT
	rCal : REAL; // Kalibrering
	iMedelvardeSekunder : UDINT := 5;
END_VAR
VAR PERSISTENT
	{attribute 'OPC.UA.DA' := '1'}
	OPM AT %M* : REAL;//Värde handställning~wp:[unit]°C[format]0.0
END_VAR

FB_BA_TiAvrg02(
	bEn:= TRUE, 
	bEnAvrg := TRUE,
	lrIn:=INT_TO_LREAL(iDataIn), 
	udiIntval:=1, 
	udiNumOfElem:= iMedelvardeSekunder, 
	lrOut=> );

FB_BA_TiAvrg01(
	bEn:= TRUE, 
	bEnAvrg := TRUE,
	lrIn:= (FB_BA_TiAvrg02.lrOut / 10) , 
	udiIntval:=1, 
	udiNumOfElem:= iMedelvardeSekunder, 
	lrOut=> );
	
fbAlarm1(bInput:= ((FB_BA_TiAvrg01.lrOut < -50) OR (FB_BA_TiAvrg01.lrOut > 150)), tAlarmDelay:= T#3S, bAutoReset:= , bAlarmOutput=> FAULT);
	
IF M THEN
	PV := OPM;
ELSIF FAULT AND (bFaultVal AND NOT (rFaultVal = -999)) THEN
	PV := rFaultVal;
ELSE
	PV := LIMIT(-50, (LREAL_TO_REAL(FB_BA_TiAvrg01.lrOut) + rCal), 150);
END_IF

//Handställningslarm
	fbAlarm2(bInput:=M , tAlarmDelay:= , bAutoReset:=TRUE , bAlarmOutput=>AL8 );

END_FUNCTION_BLOCK

// oaksLibrary/EtherCAT Specifikt/System/fbOaksSystemEtherCAT
// Funktionsblock för systemhantering av PLC för specifikt i anläggningar där EL terminaler används istället för KL
FUNCTION_BLOCK fbOaksSystemEtherCAT
VAR_INPUT
	tSekvensstartTid1 : TIME := T#5S; //Sekvensstart 1 tid
	tSekvensstartTid2 : TIME := T#10S; //Sekvensstart 2 tid
	tSekvensstartTid3 : TIME := T#15S; //Sekvensstart 3 tid
	tSekvensstartTid4 : TIME := T#20S; //Sekvensstart 4 tid
	tSekvensstartTid5 : TIME := T#25S; //Sekvensstart 5 tid
	tSekvensstartTid6 : TIME := T#30S; //Sekvensstart 6 tid
	tSekvensstartTid7 : TIME := T#35S; //Sekvensstart 7 tid
	tSekvensstartTid8 : TIME := T#40S; //Sekvensstart 8 tid
	tSekvensstartTid9 : TIME := T#45S; //Sekvensstart 9 tid
	tSekvensstartTid10 : TIME := T#50S; //Sekvensstart 10 tid
	tSekvensstartTid11 : TIME := T#60S; //Sekvensstart 11 tid
	tSekvensstartTid12 : TIME := T#65S; //Sekvensstart 12 tid
	tSekvensstartTid13 : TIME := T#70S; //Sekvensstart 13 tid
	tSekvensstartTid14 : TIME := T#75S; //Sekvensstart 14 tid
	tSekvensstartTid15 : TIME := T#80S; //Sekvensstart 15 tid
	
	M AT %M* : BOOL; //Manuell reset av larm beräkningsfel~wp:[trendoptions]i:14400, t:1
	
END_VAR

VAR_OUTPUT
	{attribute 'OPC.UA.DA' := '1'}
	AL AT %M* : BOOL; //Kritiskt beräkningsfel i PLC (kontakta OAKS)~wp:[alarmoptions]p:1
	{attribute 'OPC.UA.DA' := '1'}
	FAULT AT %M* : BOOL; //Fel på EBUS-system (kontakta OAKS)~wp:[alarmoptions]p:1
	{attribute 'OPC.UA.DA' := '1'}
	AL8 AT %M* : BOOL; //Okänd plc-modell~wp:[alarmoptions]p:3
	{attribute 'OPC.UA.DA' := '1'}
	PV8 AT %M* : STRING; //Plc-modell~wp:
	{attribute 'OPC.UA.DA' := '1'}
	PV 		: INT; // År~wp:
	{attribute 'OPC.UA.DA' := '1'}
	PV1 	: INT; // Månad(1-12)~wp:
	{attribute 'OPC.UA.DA' := '1'}
	PV2 	: INT; // Dag (1-31)~wp:
	{attribute 'OPC.UA.DA' := '1'}
	PV3		: INT; // Veckodag (1-7)~wp:
	{attribute 'OPC.UA.DA' := '1'}
	PV4 	: INT; // Timme (0-23)~wp:
	{attribute 'OPC.UA.DA' := '1'}
	PV5 	: INT; // Minut (0-59)~wp:
	{attribute 'OPC.UA.DA' := '1'}
	PV6 	: INT; // Sekund (0-59)~wp:
	{attribute 'OPC.UA.DA' := '1'}
	PV7 AT %M* : STRING; //Datum och tid från plc~wp:
	{attribute 'OPC.UA.DA' := '1'}
//	PV9 AT %M* : STRING; //Orsak FAULT (EBUS)~wp:
	bRTCFault : BOOL;	//Fel i realtidsklocka (RTC-batteri slut samt ingen NTP-konfiguration)
END_VAR

VAR
	bInit : BOOL := FALSE;	//För uppstartsfunktioner
	
	fbHardwareModelInfo01 : fbHardwareModelInfo;
	fbAlarmfbHardwareModelInfo: fbAlarm;
	
	fbPLC_SystemTime: Tc3_BA.FB_BA_GetTime;
	stTime		: tc2_ba.TIMESTRUCT;
	FB_BA_GetTime01 : tc2_ba.FB_BA_GetTime; 
//	FB_BA_ExtTiSt01 : tc2_ba.FB_BA_ExtTiSt;	
	uiInitCyCnt : UINT := 0;	
	
	fbS_UPS_CX5130				: FB_S_UPS_CX51x0;
	fbS_UPS_CX8190				: FB_S_UPS_CX81xx;
	fbS_UPS_CX9020				: FB_S_UPS_CX9020_U900;
	
	fbR_TrigPowerFailure		: Tc2_Standard.R_TRIG;
//	fbCountPowerFailure			: Tc2_Standard.CTU;
	bResetCounterPowerFailures	: BOOL; // If TRUE the fbCountPowerFailure is reset to 0
	fbR_ResetCounter			: Tc2_Standard.R_TRIG;	
//	bBootDataLoaded				: BOOL; // If TRUE bootdata file loaded. Normal behaviour.
//	bOldBootDataLoaded			: BOOL; // IF TRUE old bootdata file is loaded. bootdata-file missing or corrupt.

	fbTonSekvensstart1  : TON; //Sekvensstart 1  global variabel sätts till true efter inställd tid
	fbTonSekvensstart2  : TON; //Sekvensstart 2  global variabel sätts till true efter inställd tid
	fbTonSekvensstart3  : TON; //Sekvensstart 3  global variabel sätts till true efter inställd tid
	fbTonSekvensstart4  : TON; //Sekvensstart 4  global variabel sätts till true efter inställd tid
	fbTonSekvensstart5  : TON; //Sekvensstart 5  global variabel sätts till true efter inställd tid
	fbTonSekvensstart6  : TON; //Sekvensstart 6  global variabel sätts till true efter inställd tid
	fbTonSekvensstart7  : TON; //Sekvensstart 7  global variabel sätts till true efter inställd tid
	fbTonSekvensstart8  : TON; //Sekvensstart 8  global variabel sätts till true efter inställd tid
	fbTonSekvensstart9  : TON; //Sekvensstart 9  global variabel sätts till true efter inställd tid
	fbTonSekvensstart10 : TON; //Sekvensstart 10 global variabel sätts till true efter inställd tid
	fbTonSekvensstart11 : TON; //Sekvensstart 11 global variabel sätts till true efter inställd tid
	fbTonSekvensstart12 : TON; //Sekvensstart 12 global variabel sätts till true efter inställd tid
	fbTonSekvensstart13 : TON; //Sekvensstart 13 global variabel sätts till true efter inställd tid
	fbTonSekvensstart14 : TON; //Sekvensstart 14 global variabel sätts till true efter inställd tid
	fbTonSekvensstart15 : TON; //Sekvensstart 15 global variabel sätts till true efter inställd tid

	fbPLC_WritePersistentData: Tc3_BA.FB_BA_WrtPersistDat;
	fbTimerWritePersistent: TON;
	bManualTrigg		: BOOL;	 // Manual trigger for writing persistent data
	fbRTrigManual: Tc2_Standard.R_TRIG;
	fbRTrigExecuted: Tc2_Standard.R_TRIG;
	 
	i : UINT;
	fbToggleEbusRead : fbToggle;
	fbGetAllSlaveStates : FB_EcGetAllSlaveStates;
    devStates : ARRAY[0..255] OF ST_EcSlaveState;
    nSlaves  : UINT := 0;
	bExecuteEbus : BOOL;
	fbEcStateAlarm : fbAlarm;
    nErrId : UDINT;
	bEcError : BOOL; 
	
	fbCheck1					: fbEdge;
	fbCheck2					: fbEdge;
	fbCheck3					: fbEdge;
	fbCheck4					: fbEdge;
	fbCheck5					: fbEdge;
	fbCheck6					: fbEdge;
	fbCheck7					: fbEdge;
	fbCheck8					: fbEdge;
	fbCheck9					: fbEdge;
	fbCheck10					: fbEdge;
	fbImplicitCheckAlarm		: fbAlarm;
	
	nEcMasterSlaveCount AT %I*  : UINT; //Länk till antalet slavar
	arrEcMasterNetId AT %I* : T_AmsNetIdArr; //Länkning till masterAmsNetID
END_VAR

VAR PERSISTENT
	dtTimeLastPowerFailure		: DT;		// Last Time Power Failure
	nNumberOfPowerFailures		: UDINT;	// Number of Power Failures since last reset of counter
	
	bActivate			: BOOL	:=TRUE;		// If TRUE cyclic writing of persistent data according to 
	nCycleTime			: TIME	:=T#24H; 	// The time cycle for writing of persistent data
	dtLastTimeExecuted	: DT	;			// Last time executed writing of persistent data
	
//	bResetKBUSAutomatically 	: BOOL	:= TRUE;	//TRUE=Automatic reset of KbusFailure, FALSE=Manual reset of Kbusfailure
//	tRetrigTime 				: TIME 	:= T#30S;	//How often Kbusreset is reactivated if the last attempt is not succesfully 
//	nMaxRetries					: INT	:= 60;		//How many retries if the automatic reset is not succesful.
	
END_VAR
VAR_INPUT PERSISTENT
	sNetId : T_AmsNetId := ''; //Skriv in AMSnetID på din EtherCAT master IO Device
END_VAR

//Sekvensstart
	fbTonSekvensstart1(IN:=TRUE , PT:=tSekvensstartTid1 , Q=>oaksgvl.bSekvensstart1 , ET=> );
	fbTonSekvensstart2(IN:=TRUE , PT:=tSekvensstartTid2 , Q=>oaksgvl.bSekvensstart2 , ET=> );
	fbTonSekvensstart3(IN:=TRUE , PT:=tSekvensstartTid3 , Q=>oaksgvl.bSekvensstart3 , ET=> );
	fbTonSekvensstart4(IN:=TRUE , PT:=tSekvensstartTid4 , Q=>oaksgvl.bSekvensstart4 , ET=> );
	fbTonSekvensstart5(IN:=TRUE , PT:=tSekvensstartTid5 , Q=>oaksgvl.bSekvensstart5 , ET=> );
	fbTonSekvensstart6(IN:=TRUE , PT:=tSekvensstartTid6 , Q=>oaksgvl.bSekvensstart6 , ET=> );
	fbTonSekvensstart7(IN:=TRUE , PT:=tSekvensstartTid7 , Q=>oaksgvl.bSekvensstart7 , ET=> );
	fbTonSekvensstart8(IN:=TRUE , PT:=tSekvensstartTid8 , Q=>oaksgvl.bSekvensstart8 , ET=> );
	fbTonSekvensstart9(IN:=TRUE , PT:=tSekvensstartTid9 , Q=>oaksgvl.bSekvensstart9 , ET=> );
	fbTonSekvensstart10(IN:=TRUE , PT:=tSekvensstartTid10 , Q=>oaksgvl.bSekvensstart10 , ET=> );
	fbTonSekvensstart11(IN:=TRUE , PT:=tSekvensstartTid11 , Q=>oaksgvl.bSekvensstart11 , ET=> );
	fbTonSekvensstart12(IN:=TRUE , PT:=tSekvensstartTid12 , Q=>oaksgvl.bSekvensstart12 , ET=> );
	fbTonSekvensstart13(IN:=TRUE , PT:=tSekvensstartTid13 , Q=>oaksgvl.bSekvensstart13 , ET=> );
	fbTonSekvensstart14(IN:=TRUE , PT:=tSekvensstartTid14 , Q=>oaksgvl.bSekvensstart14 , ET=> );
	fbTonSekvensstart15(IN:=TRUE , PT:=tSekvensstartTid15 , Q=>oaksgvl.bSekvensstart15 , ET=> );
//Slut

//Konfigurering av passiva givar-kort
	oaksGVL.fbPassiveAnalogInConfigTonReset(IN:=oaksgvl.bPassiveAnalogInConfig , PT:=T#30S , Q=> , ET=> );
	IF oaksGVL.fbPassiveAnalogInConfigTonReset.Q THEN
		oaksgvl.bPassiveAnalogInConfig := FALSE;
	END_IF
//Slut

//Realtidsklocka
	FB_BA_GetTime01(bEn :=TRUE);	
	stTime := FB_BA_GetTime01.stSysTi;
	
	IF uiInitCyCnt < 10 THEN	//Sätt larm för fel i realtidsklocka om inläst år är <2023 efter 10 cykler
		uiInitCyCnt := uiInitCyCnt + 1;
	ELSE
		bRTCFault := stTime.wYear < 2023;
	END_IF
	
	PV 	:=WORD_TO_INT (stTime.wYear); 
	oaksGVL.iYear := PV;
	PV1 :=WORD_TO_INT (stTime.wMonth);
	oaksGVL.iMonth := PV1;
	PV2 :=WORD_TO_INT (stTime.wDay);
	oaksGVL.iDay := PV2;
	PV3 :=WORD_TO_INT (stTime.wDayOfWeek);
	oaksGVL.iDayOfWeek := PV3;
	PV4 :=WORD_TO_INT (stTime.wHour);
	oaksGVL.iHour := PV4;
	PV5 :=WORD_TO_INT (stTime.wMinute);
	oaksGVL.iMinute := PV5;
	PV6 :=WORD_TO_INT (stTime.wSecond);
	oaksGVL.iSecond := PV6;
	
	oaksGVL.iHourAndMinute := (oaksGVL.iHour *100) + oaksGVL.iMinute;
	
	PV7 := CONCAT(CONCAT(CONCAT(CONCAT(CONCAT(CONCAT(CONCAT(CONCAT(CONCAT(CONCAT(INT_TO_STRING(PV),'-'),INT_TO_STRING(PV1)),'-'),INT_TO_STRING(PV2)), ' '), INT_TO_STRING(PV4)),':'),INT_TO_STRING(PV5)),':'),INT_TO_STRING(PV6));
	
//SystemTime (används av andra funktioner)
	fbPLC_SystemTime( bEn:= TRUE, sNetId:= , udiUpdRtc_sec:= , bUpdRtc:= , bRdySysTi=> , bRdyTiZoInfo=> , bRdyRTC=> , udiRemTiUpd_sec=> , stSysTi=> , stUTC=> , dtSysTi=> , dtUTC=> , udiCurrentTime_ms=> , eTiZId=> , bErr=> , sErrDescr=> );
//Slut

//Kontrollera PLC-modell, sätt larm om okänd (dvs ej stöd av Oaks)
	fbHardwareModelInfo01(strHardwareModel=> );
	
	PV8 := fbHardwareModelInfo01.strHardwareModel;
	fbAlarmfbHardwareModelInfo(bInput := 	fbHardwareModelInfo01.strHardwareModel <> 'CX8190' AND 
											fbHardwareModelInfo01.strHardwareModel <> 'CX5110-0115' AND
											fbHardwareModelInfo01.strHardwareModel <> 'CX5130-0155' AND
											fbHardwareModelInfo01.strHardwareModel <> 'CX5130-0175' AND
											fbHardwareModelInfo01.strHardwareModel <> 'CX9020-B000', 
											tAlarmDelay:=T#10S, 
											bAutoReset:=, 
											bAlarmOutput=>AL8 );
//Slut
										
//Hantering av 1-sek UPS & skrivning av persistent data
	IF fbHardwareModelInfo01.strHardwareModel = 'CX8190' THEN
		fbS_UPS_CX8190(
		sNetID:= , 
		iPLCPort:= , 
		tTimeout:= , 
		eUpsMode:= , 
		ePersistentMode:= , 
		tRecoverTime:= , 
		bPowerFailDetect=> , 
		eState=> );
		fbR_TrigPowerFailure( CLK := fbS_UPS_CX8190.bPowerFailDetect, Q=> );
	ELSIF LEFT(fbHardwareModelInfo01.strHardwareModel, 4) = 'CX51'  THEN //Hela CX5100-serien
		fbS_UPS_CX5130(
		sNetID:= , 
		iPLCPort:= , 
		iUPSPort:= , 
		tTimeout:= , 
		eUpsMode:= , 
		ePersistentMode:= , 
		tRecoverTime:= , 
		bPowerFailDetect=> , 
		eState=> );	
		fbR_TrigPowerFailure( CLK := fbS_UPS_CX5130.bPowerFailDetect, Q=> );
	ELSIF fbHardwareModelInfo01.strHardwareModel = 'CX9020-B000' THEN
		fbS_UPS_CX9020(
		sNetID:= , 
		iPLCPort:= , 
		tTimeout:= , 
		eUpsMode:= , 
		ePersistentMode:= , 
		tRecoverTime:= , 
		bPowerFailDetect=> , 
		eState=> );
		fbR_TrigPowerFailure( CLK := fbS_UPS_CX9020.bPowerFailDetect, Q=> );
	END_IF
	
	IF fbR_TrigPowerFailure.Q THEN
		dtTimeLastPowerFailure := fbPLC_SystemTime.dtSysTi;
		nNumberOfPowerFailures := nNumberOfPowerFailures +1;
	END_IF
	
	fbR_ResetCounter( CLK := bResetCounterPowerFailures , Q=> );
	
	IF fbR_ResetCounter.Q THEN
		nNumberOfPowerFailures := 0;
		bResetCounterPowerFailures := FALSE;
	END_IF
	
//Write Persistent Data
	fbTimerWritePersistent( IN := bActivate AND NOT fbTimerWritePersistent.Q, PT:=nCycleTime, Q=> , ET=> );
	
	fbRTrigManual( CLK := bManualTrigg, Q=> );
	
	IF fbRTrigManual.Q THEN bManualTrigg := FALSE; END_IF
	
	fbPLC_WritePersistentData( bStt:= fbTimerWritePersistent.Q OR fbRTrigManual.Q, udiInitSttDly_sec:= , bBusy=> , udiRemTiInitSttDly_sec=> , bErr=> , sErrDescr=> );
	
	fbRTrigExecuted( CLK := fbPLC_WritePersistentData.bBusy, Q=> );
	
	IF fbRTrigExecuted.Q THEN dtLastTimeExecuted := fbPLC_SystemTime.dtSysTi; END_IF;
//Slut

//EBUS Larmhantering
sNetId:= F_CreateAmsNetId(nIds:= arrEcMasterNetId);

fbToggleEbusRead(bStart:= TRUE, tTimeOn:= T#15S, tTimeOff:= T#1S, bOutput=> bExecuteEbus);

	fbGetAllSlaveStates(sNetId:= sNetId, pStateBuf := ADR(devStates), cbBufLen:=SIZEOF(devStates), bExecute:= bExecuteEbus);
	nSlaves := nEcMasterSlaveCount;
	nErrId := fbGetAllSlaveStates.nErrId;
	
	IF fbGetAllSlaveStates.bError THEN
		bEcError := TRUE;
	ELSE
		IF nSlaves >= 2 THEN
			FOR i := 0 TO (LIMIT(1,(nSlaves -1), 200)) DO
				IF devStates[i].deviceState <> EC_DEVICE_STATE_OP THEN 
					bEcError := TRUE;
				ELSE
					bEcError := FALSE;
				END_IF 
			END_FOR
		ELSE
			bEcError:= TRUE;
		END_IF
	END_IF 
	
	fbEcStateAlarm(bInput:= bEcError, tAlarmDelay:= T#10S, bAutoReset:= TRUE, bAlarmOutput=> FAULT);
//Slut

//Hantering av larm för Implicit-kontroller (allvarligt beräkningsfel i PLC)
	fbCheck1(anyInput := oaksGVL.udiCheckBounds, bIncr := TRUE);
	fbCheck2(anyInput := oaksGVL.udiCheckDivDInt, bIncr := TRUE);
	fbCheck3(anyInput := oaksGVL.udiCheckDivLInt, bIncr := TRUE);
	fbCheck4(anyInput := oaksGVL.udiCheckDivLReal, bIncr := TRUE);
	fbCheck5(anyInput := oaksGVL.udiCheckDivReal, bIncr := TRUE);
	fbCheck6(anyInput := oaksGVL.udiCheckLRangeSigned, bIncr := TRUE);
	fbCheck7(anyInput := oaksGVL.udiCheckLRangeUnsigned, bIncr := TRUE);
	fbCheck8(anyInput := oaksGVL.udiCheckPointer, bIncr := TRUE);
	fbCheck9(anyInput := oaksGVL.udiCheckRangeSigned, bIncr := TRUE);
	fbCheck10(anyInput := oaksGVL.udiCheckRangeUnsigned, bIncr := TRUE);
	
	fbImplicitCheckAlarm.bInput := 	fbCheck1.bEdgeF OR fbCheck2.bEdgeF OR fbCheck3.bEdgeF OR fbCheck4.bEdgeF OR fbCheck5.bEdgeF OR 
									fbCheck6.bEdgeF OR fbCheck7.bEdgeF OR fbCheck8.bEdgeF OR fbCheck9.bEdgeF OR fbCheck10.bEdgeF;
									
	fbImplicitCheckAlarm(bAutoReset := M, tAlarmDelay := T#0S, bAlarmOutput => AL);
	M := FALSE;
//Slut


bInit := TRUE;	//Sätt bInit för andra funktioner

END_FUNCTION_BLOCK

// oaksLibrary/System/fbHardwareModelInfo
// Block för att läsa ut vilken modell plc är av.
FUNCTION_BLOCK fbHardwareModelInfo
VAR	
	FB_CxGetDeviceIdentificationEx01: FB_CxGetDeviceIdentificationEx;
	fbToggle1: fbToggle; // Togglar körning av FB_CxGetDeviceIdentificationEx01
	F_TRIG01: F_TRIG; // Triggar skrivning till strHardwareModel vid avslutad körning av FB_CxGetDeviceIdentificationEx01
END_VAR
VAR_OUTPUT
	strHardwareModel : STRING; // Sträng innehållande info om plc modell (exempelvis CX8190, CX5130).
END_VAR

	fbToggle1(bStart:=TRUE , tTimeOn:=T#1S , tTimeOff:=T#1S , bOutput=> );

	FB_CxGetDeviceIdentificationEx01(
	bExecute:=fbToggle1.bOutput , 
	tTimeout:= , 
	bBusy=> , 
	bError=> , 
	nErrorID=> , 
	stDevIdent=> );
	
	F_TRIG01(CLK:=FB_CxGetDeviceIdentificationEx01.bBusy , Q=> );
	
	IF F_TRIG01.Q THEN
		strHardwareModel := FB_CxGetDeviceIdentificationEx01.stDevIdent.strHardwareModel;
	END_IF

END_FUNCTION_BLOCK

// oaksLibrary/fbEdge
(* Funktionsblock som övervakar en variabel, oavsett typ (EJ STRING), och indikerar om den förändrats. Utgång för flank och vippa (kräver reset).
	Ingångar:
		anyInput:	Variabel som ska övervakas (EJ STRING)
		bRst:		Återställer utgången bEdgeSR
		bIncr:		Övervaka endast ett ökande värde
	Utgångar:
		bEdgeF	Sätts en gång om värdet förändrats (flank)
		bEdgeSR	Sätts permanent om värdet förändrats (vippa, återställs av bRst)
		bError	Variabel som övervakas har felaktig datatyp eller är en felaktig referens (t ex variabel som ej finns)
		
*)

FUNCTION_BLOCK fbEdge
VAR_INPUT
	anyInput	: ANY;		//Värde som ska övervakas (EJ STRING)
	bRst		: BOOL;		//Återställ vippa (bEdgeSR)
	bIncr		: BOOL;		//Övervaka endast om värdet ökar
END_VAR
VAR_OUTPUT
	bEdgeF		: BOOL;		//Värde har förändrats (flank)
	bEdgeSR		: BOOL;		//Värde har förändrats (vippa)
	bError		: BOOL;		//Ej kompatibel datatyp eller felaktig referens
END_VAR
VAR
	
	pAnyBool	: POINTER TO BOOL;
	pAnyByte	: POINTER TO BYTE;
	pAnyWord	: POINTER TO WORD;
	pAnyDWord	: POINTER TO DWORD;
	pAnyLWord	: POINTER TO LWORD; 
	
	lwData		: LWORD;
	lwDataOld	: LWORD;
	
	fbSR	: SR;
	
	bInit : BOOL := FALSE;
	
END_VAR

bError := FALSE;
IF anyInput.diSize <> 0 THEN
	IF (anyInput.TypeClass = __SYSTEM.TYPE_CLASS.TYPE_BOOL) OR (anyInput.TypeClass = __SYSTEM.TYPE_CLASS.TYPE_BIT) THEN	//Enbitarsvariabler måste identifieras pga 8-bits alignment i TC3
		pAnyBool := anyInput.pValue;
		lwData := BOOL_TO_LWORD(pAnyBool^);
	ELSE	//Övriga variabler är alltid 8..64 bitar i storlek om en byte
		IF anyInput.diSize = 1 THEN
			pAnyByte := anyInput.pValue;
			lwData := pAnyByte^;
		ELSIF anyInput.diSize = 2 THEN
			pAnyWord := anyInput.pValue;
			lwData := pAnyWord^;
		ELSIF anyInput.diSize = 4 THEN
			pAnyDWord := anyInput.pValue;
			lwData := pAnyDWord^;
		ELSIF anyInput.diSize = 8 THEN
			pAnyLWord := anyInput.pValue;
			lwData := pAnyLWord^;
		ELSE
			bError := TRUE;	//Ej kompatibel datatyp (troligen sträng)
		END_IF
	END_IF;
ELSE
	bError := TRUE;
END_IF

IF bInit THEN
	bEdgeF := (NOT bIncr AND (lwData <> lwDataOld)) OR (bIncr AND (lwData > lwDataOld));	//Sätt pulsutgång
	fbSR(SET1 := bEdgeF, RESET := bRst, Q1 => bEdgeSR);		//Sätt vippa
END_IF;

lwDataOld := lwData;
bInit := TRUE;

IF bRst THEN
	bRst := FALSE;
END_IF

END_FUNCTION_BLOCK

// oaksLibrary/Familjebostäder/fbMotorRadFamiljebostader
(*
	CIRKULATIONSPUMP
	Cirkulationspump stoppas då inget värmebehov föreligger.
	värmeventil är stängd och rumstemperaturen är uppnådd samt att
	utetemperaturen är över [+10 ºC] om ”Rumskompensering” är valt, annars [+14 ºC].
	Momentant stopp vid utetemperatur över [+16 ºC].
	Stoppad pump motioneras 2 min/dygn.
*)
FUNCTION_BLOCK fbMotorRadFamiljebostader EXTENDS fbMotor
VAR_INPUT
	rOutdoorTemp : ANY; // Utetemperatur används för start/stopp Knyter man inget här används oaksGVL.rOutdoortemp
	rRoomtemp : REAL; // Rumstemperatur
	rValve : REAL; // Ventilläge värmeventil
END_VAR
VAR_IN_OUT
	fbRoomCompPoseidon01 : fbRoomCompPoseidon;
END_VAR
VAR_OUTPUT
	{attribute 'OPC.UA.DA' := '1'}
	PV4  AT %M*  : BOOL; //Startvillkor momentan utetemperatur under 5°C~wp:[trendoptions]i:14400, t:1
	{attribute 'OPC.UA.DA' := '1'}
	PV5  AT %M*  : BOOL; //Startvillk. utetemp. under inst. värde vid utekomp.~wp:[trendoptions]i:14400, t:1
	{attribute 'OPC.UA.DA' := '1'}
	PV6  AT %M*  : BOOL; //Startvillk. utetemp. under inst. värde vid rumskomp.~wp:[trendoptions]i:14400, t:1
	{attribute 'OPC.UA.DA' := '1'}
	PV  AT %M* : STRING; //Aktuellt driftläge~wp:
END_VAR
VAR
	rTempUsedMean : REAL; // Uteluftstemperatur medel
	rTempUsedMomentan : REAL; // Uteluftstemperatur
	fbPumpstoppTof : TOF;
	bTemperaturStart : BOOL;
	//itemp : int;
END_VAR
VAR_INPUT PERSISTENT
	{attribute 'OPC.UA.DA' := '1'}
	SP1 AT %M* : REAL := 14;  //Stoppa pump vid rumskomp. om momentan utetemp. över~wp:[unit]°C[format]0.0
	{attribute 'OPC.UA.DA' := '1'}
	SP2 AT %M* : REAL := 10;  //Stoppa pump vid ej rumskomp. om momentan utetemp. över~wp:[unit]°C[format]0.0
	{attribute 'OPC.UA.DA' := '1'}
	SP3 AT %M* : REAL := 19;  //Tillåt ej stopp av pump vid rumskomp. om rumstemp underskr.~wp:[unit]°C[format]0.0
	{attribute 'OPC.UA.DA' := '1'}
	SP4 AT %M* : INT := 15; //Stoppfördröjning~wp:[unit]min
END_VAR

	SUPER^();

	IF SP2 < 15 THEN // minbegränsning av stoppfördröjningstid
		SP2 := 15;
	END_IF

	//Temp select
	rTempUsedMomentan := F_GetTempToUse(rOutdoorTemp);
	
	// Startar pump om utetemp underskrider
	PV4 := rTempUsedMomentan < 5;
	PV5 := rTempUsedMomentan < SP2 AND fbRoomCompPoseidon01.mIAktuelltDriftlage() = 1;
	PV6 := rTempUsedMomentan < SP1 AND rRoomtemp >  SP3 AND fbRoomCompPoseidon01.mIAktuelltDriftlage() = 2;
	
	IF PV4 OR PV5 OR PV6 THEN 
		bTemperaturStart := TRUE;
	ELSIF rValve = 0 AND NOT PV4 AND NOT PV5 AND NOT PV6 THEN
		bTemperaturStart := FALSE;
	END_IF;
	fbPumpstoppTof(IN:=bTemperaturStart , PT:=fRealToMinute(SP4) , Q=> bStart, ET=> );
		
	PV := fbRoomCompPoseidon01.PV;

END_FUNCTION_BLOCK

// oaksLibrary/Poseidon/fbRoomCompPoseidon
FUNCTION_BLOCK fbRoomCompPoseidon
VAR_INPUT
	{attribute 'OPC.UA.DA' := '1'}
	PV1 AT %M* : REAL; //Aktuell rumsmedeltemperatur~wp:[unit]°C[format]0.0
END_VAR
VAR_OUTPUT
	{attribute 'OPC.UA.DA' := '1'}
	PV AT %M* : STRING; //Aktuellt driftläge~wp:
	{attribute 'OPC.UA.DA' := '1'}
	PV2 AT %M* : REAL; //Aktuell framledningskompensering~wp:[unit]°C[format]0.0
END_VAR
VAR
	iAktuelltDriftlage : INT; //1 = Driftfall A (rumskompensering inaktiv) || 2 = Driftfall B (rumskompensering aktiv)
	itemp : INT;
END_VAR
VAR_INPUT PERSISTENT	
	{attribute 'OPC.UA.DA' := '1'}
	Y1 AT %M* : REAL:=3; //Framledningskompensering/Rumstemperatur~wp:[unit]°C[format]0.0
	{attribute 'OPC.UA.DA' := '1'}
	Y2 AT %M* :	REAL:=2; //Framledningskompensering/Rumstemperatur~wp:[unit]°C[format]0.0
	{attribute 'OPC.UA.DA' := '1'}
	Y3 AT %M* :	REAL:=1; //Framledningskompensering/Rumstemperatur~wp:[unit]°C[format]0.0
	{attribute 'OPC.UA.DA' := '1'}
	Y4 AT %M* :	REAL:=0; //Framledningskompensering/Rumstemperatur~wp:[unit]°C[format]0.0
	{attribute 'OPC.UA.DA' := '1'}
	Y5 AT %M* :	REAL:=-1; //Framledningskompensering/Rumstemperatur~wp:[unit]°C[format]0.0
	{attribute 'OPC.UA.DA' := '1'}
	Y6 AT %M* :	REAL:=-3; //Framledningskompensering/Rumstemperatur~wp:[unit]°C[format]0.0
	{attribute 'OPC.UA.DA' := '1'}
	X1 AT %M* :	REAL:=17; //Rumstemperatur~wp:[unit]°C[format]0.0
	{attribute 'OPC.UA.DA' := '1'}
	X2 AT %M* :	REAL:=18; //Rumstemperatur~wp:[unit]°C[format]0.0
	{attribute 'OPC.UA.DA' := '1'}
	X3 AT %M* :	REAL:=19; //Rumstemperatur~wp:[unit]°C[format]0.0
	{attribute 'OPC.UA.DA' := '1'}
	X4 AT %M* :	REAL:=20;  //Rumstemperatur~wp:[unit]°C[format]0.0
	{attribute 'OPC.UA.DA' := '1'}
	X5 AT %M* :	REAL:=21; //Rumstemperatur~wp:[unit]°C[format]0.0
	{attribute 'OPC.UA.DA' := '1'}
	X6 AT %M* :	REAL:=23; //Rumstemperatur~wp:[unit]°C[format]0.0
END_VAR
VAR_INPUT PERSISTENT
	{attribute 'OPC.UA.DA' := '1'}
	SP1 AT %M* : USINT := 1; //1 = Driftfall A || 2 = Driftfall B~wp:[format]0
END_VAR

IF SP1 < 1 THEN
	SP1 := 1;
ELSIF SP1 > 2 THEN
	SP1 := 2;	
END_IF

IF SP1 = 1 THEN
	PV2 := 0;
	PV := 'Driftfall A (rumskompensering inaktiv)';
	iAktuelltDriftlage := 1;
ELSE
	PV2 := fScale6p(rX:=PV1 , Y1:= Y1, Y2:=Y2 , Y3:=Y3 , Y4:=Y4 , Y5:=Y5 , Y6:=Y6 , X1:=X1 , X2:=X2 , X3:=X3, X4:=X4 , X5:=X5 , X6:=X6 );
	PV := 'Driftfall B (rumskompensering aktiv)';
	iAktuelltDriftlage := 2;
END_IF

METHOD PUBLIC mIAktuelltDriftlage : INT
VAR_INPUT
END_VAR
mIAktuelltDriftlage := iAktuelltDriftlage;
END_METHOD

END_FUNCTION_BLOCK

// oaksLibrary/Givare/fbGeneralSensor
//OAKS AB
//2022-10-28
//Generellt analog ut block med handställningsmöjlighet för tex. givare via SX:Acura
//Möjlighet till givarfel genom att ställa min/max på ingångsvärde på rSensorValee
//OPM (rHandsetrValue) och PV (rOutput) skapas som lokala variabler i programfil.
FUNCTION_BLOCK fbGeneralSensor

VAR_INPUT
rSensorValue 				: REAL := 0; //Skalat ingångsvärde
rSensorErrorMin 			: REAL := -50; //Min. begränsning givarfel
rSensorErrorMax 			: REAL := 50; //Max. begränsning givarfel
bComError 					: BOOL := FALSE; //Eventuellt kommunikationsfel
sSensorType 				: STRING(255) := ' '; //Beskrivande text av givartyp
rHandsetValue 				: REAL; //Handställningsvärde
tSensorErrorDelay		: TIME := T#30S;
END_VAR
VAR_OUTPUT
	rOutput 				: REAL;//Utgång knyts till tagg
	{attribute 'OPC.UA.DA' := '1'}
	FAULT AT %M*			: BOOL := FALSE;//Givarfel~wp:
	{attribute 'OPC.UA.DA' := '1'}
	AL8 AT %M* 				: BOOL := FALSE; //Givare handställd~wp:[alarmoptions]p:3
	{attribute 'OPC.UA.DA' := '1'}
	PV8 AT %M* 				: STRING := ' ';//Givarinformation~wp:
END_VAR
VAR
	bSensorErrorInternal	: BOOL; //Sensorfel aktiverat 
	fbAlarm_SensorError		: fbAlarm;
	sTemp 					: STRING(255) := ' ';
END_VAR
VAR_INPUT PERSISTENT
	{attribute 'OPC.UA.DA' := '1'}
	M AT %M* 				: BOOL;//Handställning~wp:[trendoptions]i:14400, t:1
END_VAR

//Manuell utsignal
	IF M THEN
		rOutput := rHandsetValue;
	ELSE 
		rOutput := rSensorValue;
	END_IF

//Larm manuell
	AL8 := M;
	
//Givarfel
	IF (rSensorValue >= rSensorErrorMax) OR (rSensorValue <= rSensorErrorMin) THEN
		bSensorErrorInternal := TRUE;
	ELSE 
		bSensorErrorInternal := FALSE;
	END_IF

	fbAlarm_SensorError(bInput:= bSensorErrorInternal OR bComError, tAlarmDelay:= tSensorErrorDelay, bAutoReset:= TRUE, bAlarmOutput=> );
	FAULT := fbAlarm_SensorError.bAlarmOutput;

//Sensor info
	PV8 := sSensorType;

END_FUNCTION_BLOCK

// oaksLibrary/Givare/fbOutDoorTempMean
FUNCTION_BLOCK fbOutDoorTempMean EXTENDS fbPT1000
VAR_OUTPUT
	{attribute 'OPC.UA.DA' := '1'}
	PV1 AT %M*  : REAL; //Medeltemperatur~wp:[unit]°C[format]0.0[trendoptions]i:300
END_VAR
VAR
	bResetMeanTemp : BOOL; //Sätt denna till TRUE för återställning av medelvärdesberäkning.
	lrMeanInternal : LREAL;
	lrMeanInternalTemp : LREAL;
	fbPLC_SystemTime: Tc3_BA.FB_BA_GetTime;
	stTime		: tc2_ba.TIMESTRUCT;

	FB_BA_GetTime01 : tc2_ba.FB_BA_GetTime; 
	FB_BA_ExtTiSt01 : tc2_ba.FB_BA_ExtTiSt;	

	
	
	wMinute : WORD;
	fbMinuteTrig : R_TRIG;
	//iTemp : INT;
	iCounter : UINT := 4319;
	
	iAntalMinuterMedel : UINT;
	iAntalMinuterForUtrakning : UINT; //Maxbegränsar antal minuter som används för beräkning beroende på hur många minuter som finns insamlade
END_VAR
VAR PERSISTENT
	wLastMinuteOfChange : WORD;	
	{attribute 'OPC.UA.DA' := '1'}
	PV7 AT %M* : UINT;  //Antal minuter insamlade för medelvärdesberäkning (max 4320)~wp:[unit]minuter[format]0

	rArrayMean72Hours : ARRAY [0..4319] OF REAL;
END_VAR

VAR_INPUT PERSISTENT
	{attribute 'OPC.UA.DA' := '1'}
	SP1 AT %M* : UINT := 12; //Antal timmar för medelvärdesberäkning (2-72)~wp:[unit]timmar[format]0
END_VAR

	SUPER^();

	IF bResetMeanTemp THEN
		bResetMeanTemp := FALSE;
		PV7 := 2;
	END_IF

	IF SP1 > 72 THEN // Medelvärdestid maxbegränsas till 72 timmar.
		SP1 := 72;
	ELSIF SP1 < 2 THEN // Medelvärdestid minbegränsas till 2 timmar.
		SP1 := 2;
	END_IF
	
	IF SP1 <= 72 AND SP1 > 1 THEN
		 iAntalMinuterMedel := SP1 * 60;
	END_IF;


	mMean(); // Metod för att räkna ut medelvärde
	//4320 minuter = 72 timmar.
	IF iAntalMinuterForUtrakning > 2 THEN
		PV1 := LREAL_TO_REAL(lrMeanInternal) / iAntalMinuterForUtrakning; 
	END_IF;
	
	//oaksGVL.rOutdoorTemp := mPv(TRUE); //utetemp som behåller sitt senaste giltiga värde vid givarfel 
	
	oaksGVL.rOutdoorTemp := mPv(bKeepLastValidData:=TRUE, rTempToUse:= rFaultVal);	//Utetemp som behåller sitt senaste giltliga värde vid givarfel, alternativ att sätta inställbart värde
	
	IF NOT FAULT THEN 
		oaksGVL.rOutdoorTempErrorValue0 := PV; // global utetemp som ställs till 0 vid givarfel.
		oaksGVL.rOutdoorTempErrorValue150 := PV;// global utetemp som ställs till 150 vid givarfel.
	ELSE
		oaksGVL.rOutdoorTempErrorValue0 := 0; // global utetemp som ställs till 0 vid givarfel.
		oaksGVL.rOutdoorTempErrorValue150 := 150;// global utetemp som ställs till 150 vid givarfel.
	END_IF
	oaksGVL.rOutdoorTempMean := PV1; // global medel utetemp
	
	oaksGVL.bOutdoorTempSensorError := FAULT; // globalt utegivarfel

METHOD PRIVATE mMean : BOOL // metod för att sköta uträkning av medelvärde
VAR_INPUT
END_VAR
	FB_BA_GetTime01(bEn :=TRUE);	
	stTime := FB_BA_GetTime01.stSysTi;

	IF stTime.wMinute <> wLastMinuteOfChange THEN
		fbMinuteTrig(CLK := TRUE);
	ELSE
		fbMinuteTrig(CLK := FALSE);
	END_IF
	//4320 minuter - 1 = 72 timmar.
	IF fbMinuteTrig.Q THEN
		FOR iCounter:= iAntalMinuterMedel - 1 TO 1 BY -1 DO
			rArrayMean72Hours[iCounter]:=rArrayMean72Hours[iCounter-1];
		END_FOR;
		rArrayMean72Hours[0] := PV;
		wLastMinuteOfChange := stTime.wMinute;
		IF PV7 < 4320 THEN // Räknas upp för att hålla koll på antal insamlade minuter
			PV7 := PV7 +1;
		END_IF
	END_IF 
	
	lrMeanInternal := 0;
	//4320 minuter - 1 = 72 timmar.
	iAntalMinuterForUtrakning := MIN(iAntalMinuterMedel,PV7); // Max begränsar antal minuter som används för beräkning beroende på hur många minuter som finns insamlade
	FOR iCounter:= iAntalMinuterForUtrakning TO 1 BY -1 DO
		lrMeanInternalTemp := lrMeanInternal;
		lrMeanInternal:=rArrayMean72Hours[iCounter-1] + lrMeanInternalTemp;
	END_FOR;
END_METHOD

END_FUNCTION_BLOCK

// oaksLibrary/Givare/fbPT1000
// PT1000 block med möjlighet att handställa PV-värde. Larmar vid givarfel eller vid handställning.
FUNCTION_BLOCK fbPT1000
VAR_INPUT
	{attribute 'OPC.UA.DA' := '1'}
	M AT %M* : BOOL;//Handställning~wp:[trendoptions]i:14400, t:1
	(*
	  KL3208_0010_PT1000              := 0,
	  KL3208_0010_NI1000              := 1,
	  KL3208_0010_NI1000_LS           := 2,
	  KL3208_0010_NTC1K8              := 3,
	  KL3208_0010_NTC1K8_TK           := 4,
	  KL3208_0010_NTC2K2              := 5,
	  KL3208_0010_NTC3K               := 6,
	  KL3208_0010_NTC5K               := 7,
	  KL3208_0010_NTC10K              := 8,
	  KL3208_0010_NTC10KPRE           := 9,
	  KL3208_0010_NTC10K_3204         := 10,
	  KL3208_0010_NTC10KTYP2          := 11,
	  KL3208_0010_NTC10KTYP3          := 12,
	  KL3208_0010_NTC10KDALE          := 13,
	  KL3208_0010_NTC10K3A221         := 14,
	  KL3208_0010_NTC20K              := 15,
	  KL3208_0010_NTC100K             := 16,
	  KL3208_0010_Poti_Resolution_01  := 17,
	  KL3208_0010_Poti_Resolution_1_1 := 18,
  	*)
	iSensorType : E_BA_SENSOR := 0;
	(*
  KL3208_0010     := 0,
  KL320x_0000     := 1,
  KL300x          := 2,
  KL301x          := 3,
  KL302x          := 4,
  KL304x          := 5,
  KL305x          := 6,
  KL306x          := 7,
  KL3132_0000     := 8,
  KL3142_0000     := 9,
  KL3152_0000     := 10,
  KL3162_0000     := 11,
  KL3172_0000     := 12,
  KL3172_0500     := 13,
  KL3172_1000     := 14,
  KL3182_0000     := 15,
  KL3404          := 16,
  KL3464          := 17,
  KL3408          := 18,
  KL3468          := 19,
  KL3444          := 20,
  KL3454          := 21,
  KL3448          := 22,
  KL3458          := 23,
*)
	iTerminalType : E_BA_Terminal_KL := 0;
	bPt100 : BOOL := FALSE;
	bFaultVal : BOOL := FALSE; //TRUE = Behåller senaste värde vid givarfel, FALSE = 150 vid kabelbrott, 0 vid kortslutning
	rFaultVal : REAL:=-999; //Om bFaultVal är TRUE så kan man välja temperatur som skall hållas här. Väljer man inget tar den senaste värdet givaren hade innan givarfel
	//OBS Tar man bort funtkion för rFaultVal i efterhand men vill behålla senaste värde (bFaultVal = TRUE) behöver man sätta rFaultVal till -999
END_VAR
VAR_OUTPUT
	{attribute 'OPC.UA.DA' := '1'}
	PV AT %M* : REAL;//Temperatur~wp:[unit]°C[format]0.0[trendoptions]i:300
	{attribute 'OPC.UA.DA' := '1'}
	FAULT AT %M* : BOOL;//Givarfel~wp:
	{attribute 'OPC.UA.DA' := '1'}
	AL8 AT %M* : BOOL; //Givare handställd~wp:[alarmoptions]p:3:
END_VAR
VAR
	fbAlarm2 : fbAlarm; // Larm handställning
	rTemp : REAL;
	usiState AT %I*: USINT;
	iDataIn AT %I*: INT;
	usiCtrl AT %Q*: USINT;
	iDataOut AT %Q*: INT;
	FB_BA_AI01 : FB_BA_AI;
	iSensorType_KL3208_0010_NTC1K8 : E_BA_SENSOR := 3;
	FB_BA_TiAvrg01,FB_BA_TiAvrg02 : tc2_ba.FB_BA_TiAvrg;
END_VAR
VAR_INPUT PERSISTENT
	{attribute 'OPC.UA.DA' := '1'}
	OPM AT %M* : REAL;//Värde handställning~wp:[unit]°C[format]0.0
	rCal : REAL; // Kalibrering
	iMedelvardeSekunder : UDINT := 5;
END_VAR

	FB_BA_AI01(
	TI_usiState:= usiState, 
	TI_iDataIn:= iDataIn, 
	eTerminal:= iTerminalType, 
	eSensor:= iSensorType, (* 0 = pt1000, *)
	bConfigurate:= oaksgvl.bPassiveAnalogInConfig, 
	rX01:= , 
	rX02:= , 
	rY01:= , 
	rY02:= , 
	rOffset:= , 
	rSmoothingFactor:= , 
	udiDecimalPlace:= , 
	bEnLimitCtrl:= , 
	rHighLimit:= 150, 
	rLowLimit:= -50, 
	udiDelayLimitCtrl_sec:= , 
	TO_usiCtrl=> usiCtrl, 
	TO_iDataOut=> iDataOut, 
	rVal=> , 
	bWireBreak=> , 
	bShortCircuit=> , 
	bHighLimit=> , 
	bLowLimit=> , 
	bErr=> , 
	sErrDescr=> );

	FB_BA_TiAvrg01(
	bEn:= TRUE, 
	bEnAvrg := TRUE,
	lrIn:=REAL_TO_LREAL(FB_BA_AI01.rVal), 
	udiIntval:=1, 
	udiNumOfElem:= iMedelvardeSekunder, 
	lrOut=> );
	
	FB_BA_TiAvrg02(
	bEn:= TRUE, 
	bEnAvrg := TRUE,
	lrIn:=REAL_TO_LREAL(iDataIn), 
	udiIntval:=1, 
	udiNumOfElem:= iMedelvardeSekunder, 
	lrOut=> );
	
	//Handställningslarm
	fbAlarm2(bInput:=M , tAlarmDelay:= , bAutoReset:=TRUE , bAlarmOutput=>AL8 );
	
	//Skriver till PV
	PV := mPv(bKeepLastValidData:=bFaultVal, rTempToUse:= rFaultVal);	// Väljer utsignal till PV	150 vid bWireBreak och 0 vid bShortCircuit med möjlighet till att behålla senaste värde eller skriva ett eget värde vid givarfel

	FAULT := FB_BA_AI01.bWireBreak OR FB_BA_AI01.bShortCircuit;

//utetemp som behåller sitt senaste giltiga värde vid givarfel 
METHOD PROTECTED mPv : REAL
VAR_INPUT
	bKeepLastValidData : BOOL;
	rTempToUse : REAL;
END_VAR



	IF M THEN
		mPv := OPM;
	ELSIF (FB_BA_AI01.bWireBreak OR FB_BA_AI01.bShortCircuit) AND (bKeepLastValidData AND NOT (rTempToUse = -999)) THEN
		mPv:= rTempToUse;
	ELSIF FB_BA_AI01.bWireBreak AND NOT bKeepLastValidData THEN
		mPv := 150;
	ELSIF FB_BA_AI01.bShortCircuit AND NOT bKeepLastValidData THEN
		mPv := -50;
	ELSIF NOT bPt100 THEN
		mPv := LREAL_TO_REAL(FB_BA_TiAvrg01.lrOut) + rCal;
	ELSE
		rTemp := LREAL_TO_REAL(FB_BA_TiAvrg02.lrOut);
		mPv := (rTemp/10) + rCal;
	END_IF
END_METHOD

END_FUNCTION_BLOCK

// oaksLibrary/Givare/fbOutDoorTempMeanLuxLightCon
(*
	0-10V block för luxgivare med belysningsvillkor samt utetempgivare med medelvärdesberäkning
*)
FUNCTION_BLOCK fbOutDoorTempMeanLuxLightCon EXTENDS fbVoltageLuxLightCon
VAR_INPUT
	rTemperatureScaleX1 : REAL; // Ändra om det är 2-10V exempelvis. Max är 0..32767 så 2-10V = 32767 * 0.2 = 6553
	rTemperatureScaleX2 : REAL := 32767;
	rTemperatureScaleMin : REAL :=-50;
	rTemperatureScaleMax : REAL := 50;
	{attribute 'OPC.UA.DA' := '1'}
	M AT %M* : BOOL;//Handställning~wp:[trendoptions]i:14400, t:1
END_VAR
VAR_OUTPUT
	{attribute 'OPC.UA.DA' := '1'}
	FAULT AT %M* : BOOL;//Givarfel temperatur~wp:
	{attribute 'OPC.UA.DA' := '1'}
	AL7 AT %M* : BOOL; //Givare handställd~wp:[alarmoptions]p:3
	{attribute 'OPC.UA.DA' := '1'}
	PV7 AT %M* : STRING := '';  //Skalning temperaturgivare~wp:
	{attribute 'OPC.UA.DA' := '1'} 
	PV AT %M* : REAL;//Utetemperatur~wp:[unit]°C[format]0.0[trendoptions]i:300
	{attribute 'OPC.UA.DA' := '1'}
	PV1 AT %M*  : REAL; //Medeltemperatur~wp:[unit]°C[format]0.0[trendoptions]i:300
END_VAR
VAR
	bResetMeanTemp : BOOL; //Sätt denna till TRUE för återställning av medelvärdesberäkning.
	lrMeanInternal : LREAL;
	lrMeanInternalTemp : LREAL;
	fbPLC_SystemTime: Tc3_BA.FB_BA_GetTime;
	stTime		: tc2_ba.TIMESTRUCT;

	FB_BA_GetTime01 : tc2_ba.FB_BA_GetTime; 
	FB_BA_ExtTiSt01 : tc2_ba.FB_BA_ExtTiSt;	

	
	
	wMinute : WORD;
	fbMinuteTrig : R_TRIG;
	//iTemp : INT;
	iCounter : UINT := 4319;
	
	iAntalMinuterMedel : UINT;
	iAntalMinuterForUtrakning : UINT; //Maxbegränsar antal minuter som används för beräkning beroende på hur många minuter som finns insamlade
	
	usiStateTemperature AT %I*: USINT;
	iDataInTemperature AT %I*: INT;
	usiCtrlTemperature AT %Q*: USINT;
	iDataOutTemperature AT %Q*: INT;
	
	FB_BA_AI01Temperatur : FB_BA_AI;
	FB_BA_TiAvrg01Temperatur : tc2_ba.FB_BA_TiAvrg;
	sTempTemperatur : STRING;
END_VAR
VAR PERSISTENT
	wLastMinuteOfChange : WORD;	
	{attribute 'OPC.UA.DA' := '1'}
	PV6 AT %M* : UINT;  //Antal minuter insamlade för medelvärdesberäkning (max 4320)~wp:[unit]minuter[format]0

	rArrayMean72Hours : ARRAY [0..4319] OF REAL;
END_VAR

VAR_INPUT PERSISTENT
	{attribute 'OPC.UA.DA' := '1'}
	OPM AT %M* : REAL;//Värde handställning~wp:[unit]°C[format]0.0
	{attribute 'OPC.UA.DA' := '1'}
	SP1 AT %M* : UINT := 12; //Antal timmar för medelvärdesberäkning (2-72)~wp:[unit]timmar[format]0
	iMedelvardeSekunderTemperatur : UDINT := 5;
END_VAR

	SUPER^();
	sTempTemperatur := CONCAT(REAL_TO_STRING(rTemperatureScaleMin),' - '); 
	PV7 := CONCAT(sTempTemperatur,REAL_TO_STRING(rTemperatureScaleMax)); 
	FB_BA_AI01Temperatur(
	TI_usiState:= usiStateTemperature, 
	TI_iDataIn:= iDataInTemperature, 
	eTerminal:= 17, 
	eSensor:= 0, (* 0 = pt1000, *)
	bConfigurate:= , 
	rX01:=rTemperatureScaleX1 , 
	rX02:=rTemperatureScaleX2 , 
	rY01:= rTemperatureScaleMin, 
	rY02:= rTemperatureScaleMax, 
	rOffset:= , 
	rSmoothingFactor:= , 
	udiDecimalPlace:= , 
	bEnLimitCtrl:= , 
	rHighLimit:= , 
	rLowLimit:=, 
	udiDelayLimitCtrl_sec:= , 
	TO_usiCtrl=> usiCtrlTemperature, 
	TO_iDataOut=> iDataOutTemperature, 
	rVal=> , 
	bWireBreak=> , 
	bShortCircuit=> , 
	bHighLimit=> , 
	bLowLimit=> , 
	bErr=> , 
	sErrDescr=> );
	
	FB_BA_TiAvrg01Temperatur(
	bEn:= TRUE, 
	bEnAvrg := TRUE,
	lrIn:=REAL_TO_LREAL(FB_BA_AI01Temperatur.rVal), 
	udiIntval:=1, 
	udiNumOfElem:= iMedelvardeSekunderTemperatur, 
	lrOut=> );

	PV:= mPv(TRUE);
	IF bResetMeanTemp THEN
		bResetMeanTemp := FALSE;
		PV6 := 2;
	END_IF

	IF SP1 > 72 THEN // Medelvärdestid maxbegränsas till 72 timmar.
		SP1 := 72;
	ELSIF SP1 < 2 THEN // Medelvärdestid minbegränsas till 2 timmar.
		SP1 := 2;
	END_IF
	
	IF SP1 <= 72 AND SP1 > 1 THEN
		 iAntalMinuterMedel := SP1 * 60;
	END_IF;
	

	mMean(); // Metod för att räkna ut medelvärde
	//4320 minuter = 72 timmar.
	IF iAntalMinuterForUtrakning > 2 THEN
		PV1 := LREAL_TO_REAL(lrMeanInternal) / iAntalMinuterForUtrakning; 
	END_IF;
	
	oaksGVL.rOutdoorTemp := mPv(TRUE); //utetemp som behåller sitt senaste giltiga värde vid givarfel 
	
